KUKA KRL program: EPS_2_251806_MH44A_A_20260213065139.src

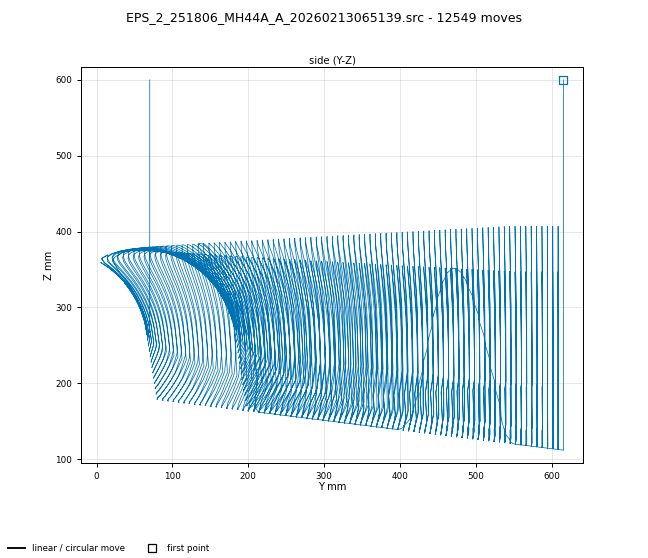
[picture p0: tool path of EPS_2_251806_MH44A_A_20260213065139.src, 12549 of 12551 moves have a stored position in this frame; points joined in program order, loops and branches not executed]
&ACCESS RVP
&REL 4
&COMMENT QRS 19112012
&PARAM EDITMASK = *
DEF PART()
EXT BAS (BAS_COMMAND :IN,REAL :IN )
INT I
BAS (#INITMOV,0 )

;KUKA QRS Post kuka4.cps  Date:22-06-2017 !

File_ID=3029

QRS_PRE_INIT()

;Init var - Until changes are made in qrs_pre_init
Outlet_Square_prg=0
Inlet_1_Square_prg=0
Inlet_2_Square_prg=0
Inlet_3_Square_prg=0
Inlet_4_Square_prg=0
Inlet_5_Square_prg=0

Outlet_1={X 0.000, Y 546.330, Z 306.500, B 0.000, E1 0.000 }
Inlet_1={X 0.000, Y 550.600, Z 246.500, B 0.000, E1 143.000 }
Outlet_1_type=201
Inlet_1_type=201
;QRS#1=Sidecore dimensions
;QRS#2=200-8" PVC SDR 35
;QRS#3=200-8" PVC SDR 35
;QRS#4=
;QRS#5=
;QRS#6=
;QRS#7=
;QRS#8=
;QRS#9=12-08 PSX
;QRS#10=12-08 PSX
;QRS#11=
;QRS#12=
;QRS#13=
;QRS#14=
;QRS#15=
;QRS#16=1220x127x686 2,25'
;QRS#17=EPS Height
;QRS#18=407
;QRS#19=*
;QRS#20= UPDATED VERSION 22-06-2017
;QRS#21=*
Outlet_Square=0100
Inlet_1_Square=0100
Inlet_2_Square=0
Inlet_3_Square=0
Inlet_4_Square=0
Inlet_5_Square=0
Mill_Square=1
Outlet_Square_Prg=204
Inlet_1_Square_prg=204

QRS_INIT()

$ADVANCE=5

; T1
PTP {E1 173.612,E2 173.612}
PTP {X 0,Y 615.492,A -85,B 0,C 180,E1 173.612,E2 173.612,E3 0,E4 0,E5 0,E6 0}
QRS_SPEED_INIT()
LIN {X 0,Y 615.492,Z 600,A -85,B 0,C 180,E1 173.612,E2 173.612,E3 0,E4 0,E5 0,E6 0} C_VEL
LIN {X 0,Y 615.492,Z 121.868,A -85,B 0,C 180,E1 173.612,E2 173.612} C_VEL
LIN {X 0,Y 615.492,Z 113.694,A -85,B 0,C 180,E1 173.612,E2 173.612} C_VEL
LIN {X 0,Y 615.479,Z 111.694,A -85,B 0,C 180,E1 173.426,E2 173.426} C_VEL
LIN {X 0,Y 615.482,Z 111.693,A -85,B 0,C 180,E1 170.801,E2 170.801} C_VEL
LIN {X 0,Y 615.486,Z 111.683,A -85,B 0,C 180,E1 168.139,E2 168.139} C_VEL
LIN {X 0,Y 615.484,Z 111.697,A -85,B 0,C 180,E1 165.451,E2 165.451} C_VEL
LIN {X 0,Y 615.48,Z 111.688,A -85,B 0,C 180,E1 162.729,E2 162.729} C_VEL
LIN {X 0,Y 615.476,Z 111.689,A -85,B 0,C 180,E1 159.967,E2 159.967} C_VEL
LIN {X 0,Y 615.483,Z 111.694,A -85,B 0,C 180,E1 157.155,E2 157.155} C_VEL
LIN {X 0,Y 615.481,Z 111.685,A -85,B 0,C 180,E1 154.284,E2 154.284} C_VEL
LIN {X 0,Y 615.497,Z 111.699,A -85,B 0,C 180,E1 151.547,E2 151.547} C_VEL
LIN {X 0,Y 615.486,Z 111.685,A -85,B 0,C 180,E1 148.914,E2 148.914} C_VEL
LIN {X 0,Y 615.481,Z 111.685,A -85,B 0,C 180,E1 146.466,E2 146.466} C_VEL
LIN {X 0,Y 615.476,Z 111.89,A -85,B 0,C 180,E1 144.275,E2 144.275} C_VEL
LIN {X 0,Y 615.459,Z 125.994,A -85,B 0,C 180,E1 141.721,E2 141.721} C_VEL
LIN {X 0,Y 615.449,Z 136.857,A -85,B 0,C 180,E1 139.801,E2 139.801} C_VEL
LIN {X 0,Y 615.471,Z 242.607,A -85,B 0,C 180,E1 138.549,E2 138.549} C_VEL
LIN {X 0,Y 615.463,Z 255.824,A -85,B 0,C 180,E1 138.261,E2 138.261} C_VEL
LIN {X 0,Y 615.479,Z 268.338,A -85,B 0,C 180,E1 137.853,E2 137.853} C_VEL
LIN {X 0,Y 615.488,Z 280.768,A -85,B 0,C 180,E1 137.3,E2 137.3} C_VEL
LIN {X 0,Y 615.491,Z 291.829,A -85,B 0,C 180,E1 136.662,E2 136.662} C_VEL
LIN {X 0,Y 615.498,Z 303.025,A -85,B 0,C 180,E1 135.852,E2 135.852} C_VEL
LIN {X 0,Y 615.498,Z 311.775,A -85,B 0,C 180,E1 135.067,E2 135.067} C_VEL
LIN {X 0,Y 615.497,Z 320.148,A -85,B 0,C 180,E1 134.148,E2 134.148} C_VEL
LIN {X 0,Y 615.496,Z 328.22,A -85,B 0,C 180,E1 133.048,E2 133.048} C_VEL
LIN {X 0,Y 615.494,Z 333.829,A -85,B 0,C 180,E1 132.081,E2 132.081} C_VEL
LIN {X 0,Y 615.494,Z 338.344,A -85,B 0,C 180,E1 131.095,E2 131.095} C_VEL
LIN {X 0,Y 615.495,Z 341.838,A -85,B 0,C 180,E1 130.09,E2 130.09} C_VEL
LIN {X 0,Y 615.495,Z 344.633,A -85,B 0,C 180,E1 128.903,E2 128.903} C_VEL
LIN {X 0,Y 615.496,Z 345.875,A -85,B 0,C 180,E1 128.013,E2 128.013} C_VEL
LIN {X 0,Y 615.493,Z 346.388,A -85,B 0,C 180,E1 126.937,E2 126.937} C_VEL
LIN {X 0,Y 615.492,Z 345.803,A -85,B 0,C 180,E1 125.834,E2 125.834} C_VEL
LIN {X 0,Y 615.496,Z 344.035,A -85,B 0,C 180,E1 124.702,E2 124.702} C_VEL
LIN {X 0,Y 615.494,Z 340.929,A -85,B 0,C 180,E1 123.535,E2 123.535} C_VEL
LIN {X 0,Y 615.496,Z 336.274,A -85,B 0,C 180,E1 122.332,E2 122.332} C_VEL
LIN {X 0,Y 615.496,Z 331.405,A -85,B 0,C 180,E1 121.385,E2 121.385} C_VEL
LIN {X 0,Y 615.493,Z 324.7,A -85,B 0,C 180,E1 120.349,E2 120.349} C_VEL
LIN {X 0,Y 615.497,Z 317.096,A -85,B 0,C 180,E1 119.406,E2 119.406} C_VEL
LIN {X 0,Y 615.499,Z 307.636,A -85,B 0,C 180,E1 118.452,E2 118.452} C_VEL
LIN {X 0,Y 615.497,Z 297.512,A -85,B 0,C 180,E1 117.637,E2 117.637} C_VEL
LIN {X 0,Y 615.468,Z 286.009,A -85,B 0,C 180,E1 116.893,E2 116.893} C_VEL
LIN {X 0,Y 615.492,Z 274.399,A -85,B 0,C 180,E1 116.307,E2 116.307} C_VEL
LIN {X 0,Y 615.485,Z 262.555,A -85,B 0,C 180,E1 115.852,E2 115.852} C_VEL
LIN {X 0,Y 615.491,Z 249.578,A -85,B 0,C 180,E1 115.497,E2 115.497} C_VEL
LIN {X 0,Y 615.492,Z 236.736,A -85,B 0,C 180,E1 115.28,E2 115.28} C_VEL
LIN {X 0,Y 615.464,Z 136.666,A -85,B 0,C 180,E1 114.105,E2 114.105} C_VEL
LIN {X 0,Y 615.49,Z 121.785,A -85,B 0,C 180,E1 111.432,E2 111.432} C_VEL
LIN {X 0,Y 615.49,Z 111.686,A -85,B 0,C 180,E1 109.598,E2 109.598} C_VEL
LIN {X 0,Y 615.468,Z 111.687,A -85,B 0,C 180,E1 107.271,E2 107.271} C_VEL
LIN {X 0,Y 615.474,Z 111.697,A -85,B 0,C 180,E1 104.549,E2 104.549} C_VEL
LIN {X 0,Y 615.488,Z 111.688,A -85,B 0,C 180,E1 101.861,E2 101.861} C_VEL
LIN {X 0,Y 615.459,Z 111.69,A -85,B 0,C 180,E1 99.199,E2 99.199} C_VEL
LIN {X 0,Y 615.492,Z 111.699,A -85,B 0,C 180,E1 96.557,E2 96.557} C_VEL
LIN {X 0,Y 615.487,Z 111.686,A -85,B 0,C 180,E1 93.928,E2 93.928} C_VEL
LIN {X 0,Y 615.459,Z 111.691,A -85,B 0,C 180,E1 91.309,E2 91.309} C_VEL
LIN {X 0,Y 615.492,Z 111.702,A -85,B 0,C 180,E1 88.691,E2 88.691} C_VEL
LIN {X 0,Y 615.486,Z 111.685,A -85,B 0,C 180,E1 86.071,E2 86.071} C_VEL
LIN {X 0,Y 615.461,Z 111.692,A -85,B 0,C 180,E1 83.443,E2 83.443} C_VEL
LIN {X 0,Y 615.492,Z 111.699,A -85,B 0,C 180,E1 80.801,E2 80.801} C_VEL
LIN {X 0,Y 615.483,Z 111.685,A -85,B 0,C 180,E1 78.139,E2 78.139} C_VEL
LIN {X 0,Y 615.466,Z 111.694,A -85,B 0,C 180,E1 75.451,E2 75.451} C_VEL
LIN {X 0,Y 615.489,Z 111.691,A -85,B 0,C 180,E1 72.73,E2 72.73} C_VEL
LIN {X 0,Y 615.465,Z 111.688,A -85,B 0,C 180,E1 69.967,E2 69.967} C_VEL
LIN {X 0,Y 615.467,Z 111.694,A -85,B 0,C 180,E1 67.659,E2 67.659} C_VEL
LIN {X 0,Y 615.488,Z 111.693,A -85,B 0,C 180,E1 65.008,E2 65.008} C_VEL
LIN {X 0,Y 615.465,Z 111.689,A -85,B 0,C 180,E1 62.084,E2 62.084} C_VEL
LIN {X 0,Y 615.468,Z 111.694,A -85,B 0,C 180,E1 59.839,E2 59.839} C_VEL
LIN {X 0,Y 615.488,Z 111.7,A -85,B 0,C 180,E1 57.543,E2 57.543} C_VEL
LIN {X 0,Y 615.488,Z 111.692,A -85,B 0,C 180,E1 55.185,E2 55.185} C_VEL
LIN {X 0,Y 615.491,Z 111.683,A -85,B 0,C 180,E1 52.758,E2 52.758} C_VEL
LIN {X 0,Y 615.475,Z 111.697,A -85,B 0,C 180,E1 49.912,E2 49.912} C_VEL
LIN {X 0,Y 615.488,Z 111.684,A -85,B 0,C 180,E1 46.952,E2 46.952} C_VEL
LIN {X 0,Y 615.469,Z 111.695,A -85,B 0,C 180,E1 44.151,E2 44.151} C_VEL
LIN {X 0,Y 615.486,Z 111.691,A -85,B 0,C 180,E1 41.474,E2 41.474} C_VEL
LIN {X 0,Y 615.48,Z 111.684,A -85,B 0,C 180,E1 38.905,E2 38.905} C_VEL
LIN {X 0,Y 615.47,Z 111.693,A -85,B 0,C 180,E1 36.426,E2 36.426} C_VEL
LIN {X 0,Y 615.486,Z 111.688,A -85,B 0,C 180,E1 33.534,E2 33.534} C_VEL
LIN {X 0,Y 615.472,Z 111.687,A -85,B 0,C 180,E1 30.92,E2 30.92} C_VEL
LIN {X 0,Y 615.479,Z 111.696,A -85,B 0,C 180,E1 28.449,E2 28.449} C_VEL
LIN {X 0,Y 615.488,Z 111.685,A -85,B 0,C 180,E1 25.57,E2 25.57} C_VEL
LIN {X 0,Y 615.47,Z 111.691,A -85,B 0,C 180,E1 22.845,E2 22.845} C_VEL
LIN {X 0,Y 615.485,Z 111.697,A -85,B 0,C 180,E1 20.557,E2 20.557} C_VEL
LIN {X 0,Y 615.484,Z 111.689,A -85,B 0,C 180,E1 17.957,E2 17.957} C_VEL
LIN {X 0,Y 615.473,Z 111.688,A -85,B 0,C 180,E1 15.226,E2 15.226} C_VEL
LIN {X 0,Y 615.49,Z 111.7,A -85,B 0,C 180,E1 12.53,E2 12.53} C_VEL
LIN {X 0,Y 615.494,Z 111.682,A -85,B 0,C 180,E1 9.862,E2 9.862} C_VEL
LIN {X 0,Y 615.472,Z 111.691,A -85,B 0,C 180,E1 7.216,E2 7.216} C_VEL
LIN {X 0,Y 615.488,Z 111.696,A -85,B 0,C 180,E1 4.584,E2 4.584} C_VEL
LIN {X 0,Y 615.5,Z 111.68,A -85,B 0,C 180,E1 1.963,E2 1.963} C_VEL
LIN {X 0,Y 615.474,Z 111.692,A -85,B 0,C 180,E1 -0.654,E2 -0.654} C_VEL
LIN {X 0,Y 615.485,Z 111.695,A -85,B 0,C 180,E1 -3.273,E2 -3.273} C_VEL
LIN {X 0,Y 615.497,Z 111.681,A -85,B 0,C 180,E1 -5.899,E2 -5.899} C_VEL
LIN {X 0,Y 615.474,Z 111.694,A -85,B 0,C 180,E1 -8.537,E2 -8.537} C_VEL
LIN {X 0,Y 615.482,Z 111.692,A -85,B 0,C 180,E1 -11.193,E2 -11.193} C_VEL
LIN {X 0,Y 615.482,Z 111.685,A -85,B 0,C 180,E1 -13.932,E2 -13.932} C_VEL
LIN {X 0,Y 615.491,Z 111.698,A -85,B 0,C 180,E1 -16.587,E2 -16.587} C_VEL
LIN {X 0,Y 615.485,Z 111.685,A -85,B 0,C 180,E1 -19.338,E2 -19.338} C_VEL
LIN {X 0,Y 615.477,Z 111.692,A -85,B 0,C 180,E1 -22.137,E2 -22.137} C_VEL
LIN {X 0,Y 615.479,Z 111.689,A -85,B 0,C 180,E1 -24.992,E2 -24.992} C_VEL
LIN {X 0,Y 615.484,Z 111.685,A -85,B 0,C 180,E1 -27.178,E2 -27.178} C_VEL
LIN {X 0,Y 615.477,Z 111.689,A -85,B 0,C 180,E1 -29.794,E2 -29.794} C_VEL
LIN {X 0,Y 615.485,Z 111.698,A -85,B 0,C 180,E1 -32.458,E2 -32.458} C_VEL
LIN {X 0,Y 615.479,Z 111.688,A -85,B 0,C 180,E1 -34.816,E2 -34.816} C_VEL
LIN {X 0,Y 615.492,Z 111.682,A -85,B 0,C 180,E1 -37.242,E2 -37.242} C_VEL
LIN {X 0,Y 615.496,Z 111.701,A -85,B 0,C 180,E1 -40.09,E2 -40.09} C_VEL
LIN {X 0,Y 615.488,Z 111.683,A -85,B 0,C 180,E1 -43.048,E2 -43.048} C_VEL
LIN {X 0,Y 615.488,Z 111.701,A -85,B 0,C 180,E1 -46.003,E2 -46.003} C_VEL
LIN {X 0,Y 615.487,Z 111.683,A -85,B 0,C 180,E1 -48.906,E2 -48.906} C_VEL
LIN {X 0,Y 615.49,Z 111.698,A -85,B 0,C 180,E1 -51.932,E2 -51.932} C_VEL
LIN {X 0,Y 615.474,Z 111.689,A -85,B 0,C 180,E1 -54.383,E2 -54.383} C_VEL
LIN {X 0,Y 615.487,Z 111.683,A -85,B 0,C 180,E1 -56.764,E2 -56.764} C_VEL
LIN {X 0,Y 615.481,Z 111.688,A -85,B 0,C 180,E1 -59.08,E2 -59.08} C_VEL
LIN {X 0,Y 615.498,Z 111.7,A -85,B 0,C 180,E1 -61.548,E2 -61.548} C_VEL
LIN {X 0,Y 615.485,Z 111.683,A -85,B 0,C 180,E1 -64.432,E2 -64.432} C_VEL
LIN {X 0,Y 615.488,Z 111.874,A -85,B 0,C 180,E1 -66.711,E2 -66.711} C_VEL
LIN {X 0,Y 615.45,Z 133.105,A -85,B 0,C 180,E1 -69.453,E2 -69.453} C_VEL
LIN {X 0,Y 615.494,Z 154.836,A -85,B 0,C 180,E1 -72.215,E2 -72.215} C_VEL
LIN {X 0,Y 615.485,Z 176.625,A -85,B 0,C 180,E1 -74.943,E2 -74.943} C_VEL
LIN {X 0,Y 615.449,Z 194.136,A -85,B 0,C 180,E1 -77.113,E2 -77.113} C_VEL
LIN {X 0,Y 615.488,Z 302.833,A -85,B 0,C 180,E1 -78.411,E2 -78.411} C_VEL
LIN {X 0,Y 615.477,Z 315.347,A -85,B 0,C 180,E1 -78.682,E2 -78.682} C_VEL
LIN {X 0,Y 615.488,Z 328.618,A -85,B 0,C 180,E1 -79.113,E2 -79.113} C_VEL
LIN {X 0,Y 615.477,Z 340.479,A -85,B 0,C 180,E1 -79.639,E2 -79.639} C_VEL
LIN {X 0,Y 615.494,Z 351.994,A -85,B 0,C 180,E1 -80.304,E2 -80.304} C_VEL
LIN {X 0,Y 615.499,Z 362.341,A -85,B 0,C 180,E1 -81.05,E2 -81.05} C_VEL
LIN {X 0,Y 615.497,Z 370.812,A -85,B 0,C 180,E1 -81.794,E2 -81.794} C_VEL
LIN {X 0,Y 615.498,Z 378.606,A -85,B 0,C 180,E1 -82.62,E2 -82.62} C_VEL
LIN {X 0,Y 615.496,Z 386.203,A -85,B 0,C 180,E1 -83.608,E2 -83.608} C_VEL
LIN {X 0,Y 615.498,Z 393.205,A -85,B 0,C 180,E1 -84.759,E2 -84.759} C_VEL
LIN {X 0,Y 615.494,Z 397.851,A -85,B 0,C 180,E1 -85.744,E2 -85.744} C_VEL
LIN {X 0,Y 615.494,Z 401.399,A -85,B 0,C 180,E1 -86.727,E2 -86.727} C_VEL
LIN {X 0,Y 615.497,Z 403.233,A -85,B 0,C 180,E1 -87.382,E2 -87.382} C_VEL
LIN {X 0,Y 615.5,Z 404.607,A -85,B 0,C 180,E1 -88.037,E2 -88.037} C_VEL
LIN {X 0,Y 615.496,Z 406.173,A -85,B 0,C 180,E1 -89.346,E2 -89.346} C_VEL
LIN {X 0,Y 615.494,Z 406.389,A -85,B 0,C 180,E1 -90,E2 -90} C_VEL
LIN {X 0,Y 615.495,Z 405.58,A -85,B 0,C 180,E1 -91.309,E2 -91.309} C_VEL
LIN {X 0,Y 615.5,Z 404.607,A -85,B 0,C 180,E1 -91.963,E2 -91.963} C_VEL
LIN {X 0,Y 615.497,Z 403.233,A -85,B 0,C 180,E1 -92.618,E2 -92.618} C_VEL
LIN {X 0,Y 615.496,Z 400.35,A -85,B 0,C 180,E1 -93.601,E2 -93.601} C_VEL
LIN {X 0,Y 615.498,Z 396.442,A -85,B 0,C 180,E1 -94.584,E2 -94.584} C_VEL
LIN {X 0,Y 615.499,Z 391.405,A -85,B 0,C 180,E1 -95.57,E2 -95.57} C_VEL
LIN {X 0,Y 615.497,Z 384.87,A -85,B 0,C 180,E1 -96.583,E2 -96.583} C_VEL
LIN {X 0,Y 615.497,Z 377.134,A -85,B 0,C 180,E1 -97.545,E2 -97.545} C_VEL
LIN {X 0,Y 615.498,Z 369.046,A -85,B 0,C 180,E1 -98.371,E2 -98.371} C_VEL
LIN {X 0,Y 615.499,Z 359.169,A -85,B 0,C 180,E1 -99.199,E2 -99.199} C_VEL
LIN {X 0,Y 615.488,Z 347.983,A -85,B 0,C 180,E1 -99.945,E2 -99.945} C_VEL
LIN {X 0,Y 615.482,Z 337.025,A -85,B 0,C 180,E1 -100.527,E2 -100.527} C_VEL
LIN {X 0,Y 615.48,Z 324.492,A -85,B 0,C 180,E1 -101.04,E2 -101.04} C_VEL
LIN {X 0,Y 615.479,Z 312.071,A -85,B 0,C 180,E1 -101.402,E2 -101.402} C_VEL
LIN {X 0,Y 615.493,Z 298.472,A -85,B 0,C 180,E1 -101.652,E2 -101.652} C_VEL
LIN {X 0,Y 615.449,Z 194.137,A -85,B 0,C 180,E1 -102.887,E2 -102.887} C_VEL
LIN {X 0,Y 615.493,Z 171.176,A -85,B 0,C 180,E1 -105.735,E2 -105.735} C_VEL
LIN {X 0,Y 615.469,Z 149.687,A -85,B 0,C 180,E1 -108.436,E2 -108.436} C_VEL
LIN {X 0,Y 615.496,Z 127.568,A -85,B 0,C 180,E1 -111.256,E2 -111.256} C_VEL
LIN {X 0,Y 615.49,Z 111.683,A -85,B 0,C 180,E1 -113.333,E2 -113.333} C_VEL
LIN {X 0,Y 615.48,Z 111.685,A -85,B 0,C 180,E1 -115.716,E2 -115.716} C_VEL
LIN {X 0,Y 615.497,Z 111.701,A -85,B 0,C 180,E1 -118.451,E2 -118.451} C_VEL
LIN {X 0,Y 615.486,Z 111.685,A -85,B 0,C 180,E1 -121.085,E2 -121.085} C_VEL
LIN {X 0,Y 615.48,Z 111.685,A -85,B 0,C 180,E1 -123.533,E2 -123.533} C_VEL
LIN {X 0,Y 615.489,Z 111.697,A -85,B 0,C 180,E1 -126.424,E2 -126.424} C_VEL
LIN {X 0,Y 615.495,Z 111.681,A -85,B 0,C 180,E1 -129.063,E2 -129.063} C_VEL
LIN {X 0,Y 615.495,Z 111.699,A -85,B 0,C 180,E1 -132.081,E2 -132.081} C_VEL
LIN {X 0,Y 615.494,Z 111.681,A -85,B 0,C 180,E1 -135.068,E2 -135.068} C_VEL
LIN {X 0,Y 615.489,Z 111.699,A -85,B 0,C 180,E1 -137.919,E2 -137.919} C_VEL
LIN {X 0,Y 615.494,Z 111.681,A -85,B 0,C 180,E1 -140.937,E2 -140.937} C_VEL
LIN {X 0,Y 615.479,Z 111.694,A -85,B 0,C 180,E1 -143.574,E2 -143.574} C_VEL
LIN {X 0,Y 615.484,Z 111.686,A -85,B 0,C 180,E1 -146.466,E2 -146.466} C_VEL
LIN {X 0,Y 615.476,Z 111.687,A -85,B 0,C 180,E1 -149.079,E2 -149.079} C_VEL
LIN {X 0,Y 615.488,Z 111.697,A -85,B 0,C 180,E1 -151.549,E2 -151.549} C_VEL
LIN {X 0,Y 615.486,Z 111.684,A -85,B 0,C 180,E1 -154.431,E2 -154.431} C_VEL
LIN {X 0,Y 615.474,Z 111.693,A -85,B 0,C 180,E1 -157.155,E2 -157.155} C_VEL
LIN {X 0,Y 615.492,Z 111.699,A -85,B 0,C 180,E1 -159.441,E2 -159.441} C_VEL
LIN {X 0,Y 615.479,Z 111.688,A -85,B 0,C 180,E1 -162.043,E2 -162.043} C_VEL
LIN {X 0,Y 615.476,Z 111.688,A -85,B 0,C 180,E1 -164.774,E2 -164.774} C_VEL
LIN {X 0,Y 615.491,Z 111.697,A -85,B 0,C 180,E1 -167.47,E2 -167.47} C_VEL
LIN {X 0,Y 615.494,Z 111.682,A -85,B 0,C 180,E1 -170.138,E2 -170.138} C_VEL
LIN {X 0,Y 615.476,Z 111.692,A -85,B 0,C 180,E1 -172.784,E2 -172.784} C_VEL
LIN {X 0,Y 615.485,Z 111.695,A -85,B 0,C 180,E1 -175.415,E2 -175.415} C_VEL
LIN {X 0,Y 615.5,Z 111.68,A -85,B 0,C 180,E1 -178.037,E2 -178.037} C_VEL
LIN {X 0,Y 615.475,Z 111.693,A -85,B 0,C 180,E1 -180.654,E2 -180.654} C_VEL
LIN {X 0,Y 615.483,Z 111.694,A -85,B 0,C 180,E1 -183.273,E2 -183.273} C_VEL
LIN {X 0,Y 615.497,Z 111.68,A -85,B 0,C 180,E1 -185.898,E2 -185.898} C_VEL
LIN {X 0,Y 615.479,Z 111.694,A -85,B 0,C 180,E1 -186.574,E2 -186.574} C_VEL
LIN {X 0,Y 614.805,Z 111.843,A -85,B 0,C 180,E1 -187.12,E2 -187.12} C_VEL
LIN {X 0,Y 611.97,Z 112.249,A -85,B 0,C 180,E1 -188.006,E2 -188.006} C_VEL
LIN {X 0,Y 609.579,Z 112.562,A -85,B 0,C 180,E1 -188.719,E2 -188.719} C_VEL
LIN {X 0,Y 608.547,Z 112.68,A -85,B 0,C 180,E1 -189.269,E2 -189.269} C_VEL
LIN {X 0,Y 608.459,Z 112.688,A -85,B 0,C 180,E1 -189.455,E2 -189.455} C_VEL
LIN {X 0,Y 608.46,Z 112.687,A -85,B 0,C 180,E1 -192,E2 -192} C_VEL
LIN {X 0,Y 608.472,Z 112.696,A -85,B 0,C 180,E1 -194.72,E2 -194.72} C_VEL
LIN {X 0,Y 608.446,Z 112.689,A -85,B 0,C 180,E1 -197.477,E2 -197.477} C_VEL
LIN {X 0,Y 608.458,Z 112.692,A -85,B 0,C 180,E1 -200.274,E2 -200.274} C_VEL
LIN {X 0,Y 608.456,Z 112.697,A -85,B 0,C 180,E1 -202.476,E2 -202.476} C_VEL
LIN {X 0,Y 608.449,Z 112.688,A -85,B 0,C 180,E1 -205.301,E2 -205.301} C_VEL
LIN {X 0,Y 608.444,Z 112.689,A -85,B 0,C 180,E1 -207.518,E2 -207.518} C_VEL
LIN {X 0,Y 608.459,Z 112.691,A -85,B 0,C 180,E1 -209.971,E2 -209.971} C_VEL
LIN {X 0,Y 608.464,Z 112.693,A -85,B 0,C 180,E1 -212.523,E2 -212.523} C_VEL
LIN {X 0,Y 608.436,Z 112.69,A -85,B 0,C 180,E1 -215.278,E2 -215.278} C_VEL
LIN {X 0,Y 608.469,Z 112.882,A -85,B 0,C 180,E1 -215.682,E2 -215.682} C_VEL
LIN {X 0,Y 608.454,Z 126.888,A -85,B 0,C 180,E1 -218.239,E2 -218.239} C_VEL
LIN {X 0,Y 608.41,Z 136.835,A -85,B 0,C 180,E1 -220.036,E2 -220.036} C_VEL
LIN {X 0,Y 608.566,Z 209.469,A -85,B 0,C 180,E1 -220.911,E2 -220.911} C_VEL
LIN {X 0,Y 608.527,Z 243.725,A -85,B 0,C 180,E1 -221.336,E2 -221.336} C_VEL
LIN {X 0,Y 608.498,Z 257.197,A -85,B 0,C 180,E1 -221.643,E2 -221.643} C_VEL
LIN {X 0,Y 608.518,Z 269.405,A -85,B 0,C 180,E1 -222.056,E2 -222.056} C_VEL
LIN {X 0,Y 608.498,Z 281.583,A -85,B 0,C 180,E1 -222.615,E2 -222.615} C_VEL
LIN {X 0,Y 608.481,Z 293.329,A -85,B 0,C 180,E1 -223.31,E2 -223.31} C_VEL
LIN {X 0,Y 608.471,Z 303.556,A -85,B 0,C 180,E1 -224.067,E2 -224.067} C_VEL
LIN {X 0,Y 608.459,Z 313.651,A -85,B 0,C 180,E1 -225,E2 -225} C_VEL
LIN {X 0,Y 608.465,Z 321.857,A -85,B 0,C 180,E1 -225.933,E2 -225.933} C_VEL
LIN {X 0,Y 608.448,Z 328.564,A -85,B 0,C 180,E1 -226.868,E2 -226.868} C_VEL
LIN {X 0,Y 608.429,Z 334.691,A -85,B 0,C 180,E1 -227.936,E2 -227.936} C_VEL
LIN {X 0,Y 608.431,Z 338.725,A -85,B 0,C 180,E1 -228.822,E2 -228.822} C_VEL
LIN {X 0,Y 608.435,Z 343.094,A -85,B 0,C 180,E1 -230.128,E2 -230.128} C_VEL
LIN {X 0,Y 608.415,Z 345.781,A -85,B 0,C 180,E1 -231.408,E2 -231.408} C_VEL
LIN {X 0,Y 608.428,Z 346.691,A -85,B 0,C 180,E1 -232.251,E2 -232.251} C_VEL
LIN {X 0,Y 608.429,Z 346.997,A -85,B 0,C 180,E1 -233.084,E2 -233.084} C_VEL
LIN {X 0,Y 608.42,Z 346.607,A -85,B 0,C 180,E1 -233.958,E2 -233.958} C_VEL
LIN {X 0,Y 608.423,Z 345.089,A -85,B 0,C 180,E1 -235.098,E2 -235.098} C_VEL
LIN {X 0,Y 608.435,Z 342.045,A -85,B 0,C 180,E1 -236.328,E2 -236.328} C_VEL
LIN {X 0,Y 608.428,Z 337.808,A -85,B 0,C 180,E1 -237.482,E2 -237.482} C_VEL
LIN {X 0,Y 608.453,Z 331.568,A -85,B 0,C 180,E1 -238.731,E2 -238.731} C_VEL
LIN {X 0,Y 608.444,Z 324.761,A -85,B 0,C 180,E1 -239.774,E2 -239.774} C_VEL
LIN {X 0,Y 608.451,Z 316.481,A -85,B 0,C 180,E1 -240.79,E2 -240.79} C_VEL
LIN {X 0,Y 608.467,Z 306.918,A -85,B 0,C 180,E1 -241.734,E2 -241.734} C_VEL
LIN {X 0,Y 608.479,Z 296.237,A -85,B 0,C 180,E1 -242.58,E2 -242.58} C_VEL
LIN {X 0,Y 608.464,Z 286.143,A -85,B 0,C 180,E1 -243.227,E2 -243.227} C_VEL
LIN {X 0,Y 608.509,Z 274.25,A -85,B 0,C 180,E1 -243.829,E2 -243.829} C_VEL
LIN {X 0,Y 608.524,Z 261.875,A -85,B 0,C 180,E1 -244.303,E2 -244.303} C_VEL
LIN {X 0,Y 608.549,Z 249.13,A -85,B 0,C 180,E1 -244.649,E2 -244.649} C_VEL
LIN {X 0,Y 608.55,Z 236.184,A -85,B 0,C 180,E1 -244.864,E2 -244.864} C_VEL
LIN {X 0,Y 608.43,Z 136.897,A -85,B 0,C 180,E1 -246.042,E2 -246.042} C_VEL
LIN {X 0,Y 608.485,Z 122.406,A -85,B 0,C 180,E1 -248.665,E2 -248.665} C_VEL
LIN {X 0,Y 608.472,Z 112.687,A -85,B 0,C 180,E1 -250.474,E2 -250.474} C_VEL
LIN {X 0,Y 608.469,Z 112.691,A -85,B 0,C 180,E1 -253.471,E2 -253.471} C_VEL
LIN {X 0,Y 608.476,Z 112.69,A -85,B 0,C 180,E1 -255.98,E2 -255.98} C_VEL
LIN {X 0,Y 608.432,Z 112.69,A -85,B 0,C 180,E1 -258.676,E2 -258.676} C_VEL
LIN {X 0,Y 608.45,Z 112.695,A -85,B 0,C 180,E1 -261.364,E2 -261.364} C_VEL
LIN {X 0,Y 608.494,Z 112.685,A -85,B 0,C 180,E1 -264.033,E2 -264.033} C_VEL
LIN {X 0,Y 608.454,Z 112.688,A -85,B 0,C 180,E1 -266.689,E2 -266.689} C_VEL
LIN {X 0,Y 608.481,Z 112.694,A -85,B 0,C 180,E1 -269.338,E2 -269.338} C_VEL
LIN {X 0,Y 608.469,Z 112.687,A -85,B 0,C 180,E1 -271.986,E2 -271.986} C_VEL
LIN {X 0,Y 608.432,Z 112.692,A -85,B 0,C 180,E1 -274.638,E2 -274.638} C_VEL
LIN {X 0,Y 608.432,Z 112.692,A -85,B 0,C 180,E1 -276.633,E2 -276.633} C_VEL
LIN {X 0,Y 608.475,Z 112.692,A -85,B 0,C 180,E1 -279.306,E2 -279.306} C_VEL
LIN {X 0,Y 608.455,Z 112.687,A -85,B 0,C 180,E1 -282,E2 -282} C_VEL
LIN {X 0,Y 608.464,Z 112.692,A -85,B 0,C 180,E1 -284.721,E2 -284.721} C_VEL
LIN {X 0,Y 608.45,Z 112.69,A -85,B 0,C 180,E1 -287.477,E2 -287.477} C_VEL
LIN {X 0,Y 608.448,Z 112.69,A -85,B 0,C 180,E1 -290.275,E2 -290.275} C_VEL
LIN {X 0,Y 608.459,Z 112.692,A -85,B 0,C 180,E1 -292.476,E2 -292.476} C_VEL
LIN {X 0,Y 608.451,Z 112.69,A -85,B 0,C 180,E1 -295.301,E2 -295.301} C_VEL
LIN {X 0,Y 608.443,Z 112.689,A -85,B 0,C 180,E1 -297.518,E2 -297.518} C_VEL
LIN {X 0,Y 608.451,Z 112.689,A -85,B 0,C 180,E1 -299.969,E2 -299.969} C_VEL
LIN {X 0,Y 608.462,Z 112.697,A -85,B 0,C 180,E1 -302.523,E2 -302.523} C_VEL
LIN {X 0,Y 608.435,Z 112.69,A -85,B 0,C 180,E1 -305.278,E2 -305.278} C_VEL
LIN {X 0,Y 608.461,Z 112.688,A -85,B 0,C 180,E1 -307.747,E2 -307.747} C_VEL
LIN {X 0,Y 608.447,Z 112.699,A -85,B 0,C 180,E1 -310.329,E2 -310.329} C_VEL
LIN {X 0,Y 608.456,Z 112.688,A -85,B 0,C 180,E1 -312.959,E2 -312.959} C_VEL
LIN {X 0,Y 608.443,Z 112.692,A -85,B 0,C 180,E1 -315.737,E2 -315.737} C_VEL
LIN {X 0,Y 608.459,Z 112.693,A -85,B 0,C 180,E1 -317.939,E2 -317.939} C_VEL
LIN {X 0,Y 608.479,Z 112.686,A -85,B 0,C 180,E1 -320.701,E2 -320.701} C_VEL
LIN {X 0,Y 608.45,Z 112.688,A -85,B 0,C 180,E1 -323.085,E2 -323.085} C_VEL
LIN {X 0,Y 608.461,Z 112.69,A -85,B 0,C 180,E1 -325.53,E2 -325.53} C_VEL
LIN {X 0,Y 608.462,Z 112.697,A -85,B 0,C 180,E1 -327.905,E2 -327.905} C_VEL
LIN {X 0,Y 608.469,Z 112.69,A -85,B 0,C 180,E1 -330.221,E2 -330.221} C_VEL
LIN {X 0,Y 608.472,Z 112.685,A -85,B 0,C 180,E1 -332.793,E2 -332.793} C_VEL
LIN {X 0,Y 608.449,Z 112.694,A -85,B 0,C 180,E1 -335.429,E2 -335.429} C_VEL
LIN {X 0,Y 608.472,Z 112.686,A -85,B 0,C 180,E1 -338.309,E2 -338.309} C_VEL
LIN {X 0,Y 608.469,Z 112.691,A -85,B 0,C 180,E1 -341.284,E2 -341.284} C_VEL
LIN {X 0,Y 608.461,Z 112.69,A -85,B 0,C 180,E1 -343.906,E2 -343.906} C_VEL
LIN {X 0,Y 608.454,Z 112.688,A -85,B 0,C 180,E1 -346.643,E2 -346.643} C_VEL
LIN {X 0,Y 608.463,Z 112.697,A -85,B 0,C 180,E1 -349.35,E2 -349.35} C_VEL
LIN {X 0,Y 608.479,Z 112.685,A -85,B 0,C 180,E1 -352.033,E2 -352.033} C_VEL
LIN {X 0,Y 608.454,Z 112.69,A -85,B 0,C 180,E1 -354.698,E2 -354.698} C_VEL
LIN {X 0,Y 608.473,Z 112.692,A -85,B 0,C 180,E1 -357.352,E2 -357.352} C_VEL
LIN {X 0,Y 608.477,Z 112.685,A -85,B 0,C 180,E1 -360,E2 -360} C_VEL
LIN {X 0,Y 608.467,Z 112.69,A -85,B 0,C 180,E1 -362.648,E2 -362.648} C_VEL
LIN {X 0,Y 608.464,Z 112.691,A -85,B 0,C 180,E1 -365.302,E2 -365.302} C_VEL
LIN {X 0,Y 608.476,Z 112.685,A -85,B 0,C 180,E1 -367.967,E2 -367.967} C_VEL
LIN {X 0,Y 608.461,Z 112.694,A -85,B 0,C 180,E1 -370.65,E2 -370.65} C_VEL
LIN {X 0,Y 608.46,Z 112.688,A -85,B 0,C 180,E1 -373.357,E2 -373.357} C_VEL
LIN {X 0,Y 608.457,Z 112.689,A -85,B 0,C 180,E1 -376.094,E2 -376.094} C_VEL
LIN {X 0,Y 608.457,Z 112.693,A -85,B 0,C 180,E1 -378.87,E2 -378.87} C_VEL
LIN {X 0,Y 608.469,Z 112.686,A -85,B 0,C 180,E1 -381.692,E2 -381.692} C_VEL
LIN {X 0,Y 608.45,Z 112.697,A -85,B 0,C 180,E1 -384.571,E2 -384.571} C_VEL
LIN {X 0,Y 608.477,Z 112.685,A -85,B 0,C 180,E1 -387.208,E2 -387.208} C_VEL
LIN {X 0,Y 608.462,Z 112.691,A -85,B 0,C 180,E1 -389.971,E2 -389.971} C_VEL
LIN {X 0,Y 608.458,Z 112.689,A -85,B 0,C 180,E1 -392.88,E2 -392.88} C_VEL
LIN {X 0,Y 608.436,Z 112.69,A -85,B 0,C 180,E1 -395.278,E2 -395.278} C_VEL
LIN {X 0,Y 608.473,Z 112.689,A -85,B 0,C 180,E1 -397.746,E2 -397.746} C_VEL
LIN {X 0,Y 608.453,Z 112.694,A -85,B 0,C 180,E1 -400.329,E2 -400.329} C_VEL
LIN {X 0,Y 608.454,Z 112.687,A -85,B 0,C 180,E1 -402.96,E2 -402.96} C_VEL
LIN {X 0,Y 608.461,Z 112.693,A -85,B 0,C 180,E1 -405.736,E2 -405.736} C_VEL
LIN {X 0,Y 608.458,Z 112.687,A -85,B 0,C 180,E1 -408.659,E2 -408.659} C_VEL
LIN {X 0,Y 608.47,Z 112.689,A -85,B 0,C 180,E1 -411.412,E2 -411.412} C_VEL
LIN {X 0,Y 608.446,Z 112.695,A -85,B 0,C 180,E1 -413.955,E2 -413.955} C_VEL
LIN {X 0,Y 608.448,Z 112.69,A -85,B 0,C 180,E1 -416.329,E2 -416.329} C_VEL
LIN {X 0,Y 608.448,Z 112.688,A -85,B 0,C 180,E1 -418.733,E2 -418.733} C_VEL
LIN {X 0,Y 608.478,Z 112.692,A -85,B 0,C 180,E1 -421.38,E2 -421.38} C_VEL
LIN {X 0,Y 608.468,Z 112.686,A -85,B 0,C 180,E1 -424.28,E2 -424.28} C_VEL
LIN {X 0,Y 608.467,Z 112.727,A -85,B 0,C 180,E1 -426.539,E2 -426.539} C_VEL
LIN {X 0,Y 608.595,Z 127.568,A -85,B 0,C 180,E1 -428.491,E2 -428.491} C_VEL
LIN {X 0,Y 608.498,Z 149.174,A -85,B 0,C 180,E1 -431.277,E2 -431.277} C_VEL
LIN {X 0,Y 608.495,Z 168.579,A -85,B 0,C 180,E1 -433.744,E2 -433.744} C_VEL
LIN {X 0,Y 608.479,Z 190.346,A -85,B 0,C 180,E1 -436.474,E2 -436.474} C_VEL
LIN {X 0,Y 608.446,Z 194.355,A -85,B 0,C 180,E1 -436.972,E2 -436.972} C_VEL
LIN {X 0,Y 608.546,Z 302.949,A -85,B 0,C 180,E1 -438.277,E2 -438.277} C_VEL
LIN {X 0,Y 608.512,Z 316.218,A -85,B 0,C 180,E1 -438.572,E2 -438.572} C_VEL
LIN {X 0,Y 608.514,Z 328.629,A -85,B 0,C 180,E1 -438.982,E2 -438.982} C_VEL
LIN {X 0,Y 608.499,Z 340.635,A -85,B 0,C 180,E1 -439.519,E2 -439.519} C_VEL
LIN {X 0,Y 608.484,Z 352.198,A -85,B 0,C 180,E1 -440.191,E2 -440.191} C_VEL
LIN {X 0,Y 608.485,Z 362.594,A -85,B 0,C 180,E1 -440.946,E2 -440.946} C_VEL
LIN {X 0,Y 608.475,Z 371.112,A -85,B 0,C 180,E1 -441.699,E2 -441.699} C_VEL
LIN {X 0,Y 608.471,Z 378.96,A -85,B 0,C 180,E1 -442.534,E2 -442.534} C_VEL
LIN {X 0,Y 608.461,Z 386.287,A -85,B 0,C 180,E1 -443.485,E2 -443.485} C_VEL
LIN {X 0,Y 608.451,Z 391.866,A -85,B 0,C 180,E1 -444.366,E2 -444.366} C_VEL
LIN {X 0,Y 608.432,Z 396.95,A -85,B 0,C 180,E1 -445.362,E2 -445.362} C_VEL
LIN {X 0,Y 608.449,Z 400.896,A -85,B 0,C 180,E1 -446.358,E2 -446.358} C_VEL
LIN {X 0,Y 608.425,Z 403.809,A -85,B 0,C 180,E1 -447.352,E2 -447.352} C_VEL
LIN {X 0,Y 608.445,Z 405.201,A -85,B 0,C 180,E1 -448.014,E2 -448.014} C_VEL
LIN {X 0,Y 608.438,Z 406.783,A -85,B 0,C 180,E1 -449.338,E2 -449.338} C_VEL
LIN {X 0,Y 608.434,Z 407,A -85,B 0,C 180,E1 -450,E2 -450} C_VEL
LIN {X 0,Y 608.448,Z 406.184,A -85,B 0,C 180,E1 -451.324,E2 -451.324} C_VEL
LIN {X 0,Y 608.445,Z 405.201,A -85,B 0,C 180,E1 -451.986,E2 -451.986} C_VEL
LIN {X 0,Y 608.425,Z 403.809,A -85,B 0,C 180,E1 -452.648,E2 -452.648} C_VEL
LIN {X 0,Y 608.449,Z 400.896,A -85,B 0,C 180,E1 -453.642,E2 -453.642} C_VEL
LIN {X 0,Y 608.432,Z 396.95,A -85,B 0,C 180,E1 -454.638,E2 -454.638} C_VEL
LIN {X 0,Y 608.438,Z 390.877,A -85,B 0,C 180,E1 -455.801,E2 -455.801} C_VEL
LIN {X 0,Y 608.462,Z 384.236,A -85,B 0,C 180,E1 -456.799,E2 -456.799} C_VEL
LIN {X 0,Y 608.456,Z 375.99,A -85,B 0,C 180,E1 -457.8,E2 -457.8} C_VEL
LIN {X 0,Y 608.472,Z 367.537,A -85,B 0,C 180,E1 -458.636,E2 -458.636} C_VEL
LIN {X 0,Y 608.479,Z 357.092,A -85,B 0,C 180,E1 -459.473,E2 -459.473} C_VEL
LIN {X 0,Y 608.489,Z 346.758,A -85,B 0,C 180,E1 -460.145,E2 -460.145} C_VEL
LIN {X 0,Y 608.519,Z 335.268,A -85,B 0,C 180,E1 -460.74,E2 -460.74} C_VEL
LIN {X 0,Y 608.528,Z 322.893,A -85,B 0,C 180,E1 -461.225,E2 -461.225} C_VEL
LIN {X 0,Y 608.544,Z 309.443,A -85,B 0,C 180,E1 -461.597,E2 -461.597} C_VEL
LIN {X 0,Y 608.552,Z 297.092,A -85,B 0,C 180,E1 -461.808,E2 -461.808} C_VEL
LIN {X 0,Y 608.434,Z 194.27,A -85,B 0,C 180,E1 -463.038,E2 -463.038} C_VEL
LIN {X 0,Y 608.523,Z 171.24,A -85,B 0,C 180,E1 -465.92,E2 -465.92} C_VEL
LIN {X 0,Y 608.53,Z 150.97,A -85,B 0,C 180,E1 -468.492,E2 -468.492} C_VEL
LIN {X 0,Y 608.571,Z 130.298,A -85,B 0,C 180,E1 -471.154,E2 -471.154} C_VEL
LIN {X 0,Y 608.52,Z 112.898,A -85,B 0,C 180,E1 -473.436,E2 -473.436} C_VEL
LIN {X 0,Y 608.459,Z 112.69,A -85,B 0,C 180,E1 -473.845,E2 -473.845} C_VEL
LIN {X 0,Y 608.443,Z 112.692,A -85,B 0,C 180,E1 -476.035,E2 -476.035} C_VEL
LIN {X 0,Y 608.477,Z 112.692,A -85,B 0,C 180,E1 -478.62,E2 -478.62} C_VEL
LIN {X 0,Y 608.446,Z 112.688,A -85,B 0,C 180,E1 -481.317,E2 -481.317} C_VEL
LIN {X 0,Y 608.473,Z 112.687,A -85,B 0,C 180,E1 -483.735,E2 -483.735} C_VEL
LIN {X 0,Y 608.446,Z 112.696,A -85,B 0,C 180,E1 -486.092,E2 -486.092} C_VEL
LIN {X 0,Y 608.47,Z 112.69,A -85,B 0,C 180,E1 -488.588,E2 -488.588} C_VEL
LIN {X 0,Y 608.457,Z 112.687,A -85,B 0,C 180,E1 -491.341,E2 -491.341} C_VEL
LIN {X 0,Y 608.464,Z 112.694,A -85,B 0,C 180,E1 -494.264,E2 -494.264} C_VEL
LIN {X 0,Y 608.453,Z 112.687,A -85,B 0,C 180,E1 -497.04,E2 -497.04} C_VEL
LIN {X 0,Y 608.452,Z 112.693,A -85,B 0,C 180,E1 -499.696,E2 -499.696} C_VEL
LIN {X 0,Y 608.471,Z 112.69,A -85,B 0,C 180,E1 -502.254,E2 -502.254} C_VEL
LIN {X 0,Y 608.442,Z 112.689,A -85,B 0,C 180,E1 -505.095,E2 -505.095} C_VEL
LIN {X 0,Y 608.467,Z 112.694,A -85,B 0,C 180,E1 -507.905,E2 -507.905} C_VEL
LIN {X 0,Y 608.466,Z 112.689,A -85,B 0,C 180,E1 -510.22,E2 -510.22} C_VEL
LIN {X 0,Y 608.475,Z 112.685,A -85,B 0,C 180,E1 -512.793,E2 -512.793} C_VEL
LIN {X 0,Y 608.452,Z 112.695,A -85,B 0,C 180,E1 -515.429,E2 -515.429} C_VEL
LIN {X 0,Y 608.471,Z 112.686,A -85,B 0,C 180,E1 -518.308,E2 -518.308} C_VEL
LIN {X 0,Y 608.473,Z 112.692,A -85,B 0,C 180,E1 -521.282,E2 -521.282} C_VEL
LIN {X 0,Y 608.46,Z 112.689,A -85,B 0,C 180,E1 -523.906,E2 -523.906} C_VEL
LIN {X 0,Y 608.455,Z 112.688,A -85,B 0,C 180,E1 -526.643,E2 -526.643} C_VEL
LIN {X 0,Y 608.464,Z 112.696,A -85,B 0,C 180,E1 -529.35,E2 -529.35} C_VEL
LIN {X 0,Y 608.478,Z 112.685,A -85,B 0,C 180,E1 -532.033,E2 -532.033} C_VEL
LIN {X 0,Y 608.457,Z 112.69,A -85,B 0,C 180,E1 -534.698,E2 -534.698} C_VEL
LIN {X 0,Y 608.475,Z 112.691,A -85,B 0,C 180,E1 -537.352,E2 -537.352} C_VEL
LIN {X 0,Y 608.477,Z 112.684,A -85,B 0,C 180,E1 -540,E2 -540} C_VEL
LIN {X 0,Y 608.469,Z 112.69,A -85,B 0,C 180,E1 -542.648,E2 -542.648} C_VEL
LIN {X 0,Y 608.463,Z 112.691,A -85,B 0,C 180,E1 -545.302,E2 -545.302} C_VEL
LIN {X 0,Y 608.476,Z 112.685,A -85,B 0,C 180,E1 -547.967,E2 -547.967} C_VEL
LIN {X 0,Y 608.459,Z 112.688,A -85,B 0,C 180,E1 -549.455,E2 -549.455} C_VEL
LIN {X 0,Y 607.783,Z 112.773,A -85,B 0,C 180,E1 -550.007,E2 -550.007} C_VEL
LIN {X 0,Y 604.929,Z 113.135,A -85,B 0,C 180,E1 -550.904,E2 -550.904} C_VEL
LIN {X 0,Y 602.524,Z 113.43,A -85,B 0,C 180,E1 -551.626,E2 -551.626} C_VEL
LIN {X 0,Y 601.491,Z 113.557,A -85,B 0,C 180,E1 -552.182,E2 -552.182} C_VEL
LIN {X 0,Y 601.407,Z 113.568,A -85,B 0,C 180,E1 -552.371,E2 -552.371} C_VEL
LIN {X 0,Y 601.426,Z 113.57,A -85,B 0,C 180,E1 -554.897,E2 -554.897} C_VEL
LIN {X 0,Y 601.431,Z 113.567,A -85,B 0,C 180,E1 -556.986,E2 -556.986} C_VEL
LIN {X 0,Y 601.402,Z 113.566,A -85,B 0,C 180,E1 -559.809,E2 -559.809} C_VEL
LIN {X 0,Y 601.413,Z 113.575,A -85,B 0,C 180,E1 -562.606,E2 -562.606} C_VEL
LIN {X 0,Y 601.4,Z 113.571,A -85,B 0,C 180,E1 -564.879,E2 -564.879} C_VEL
LIN {X 0,Y 601.419,Z 113.566,A -85,B 0,C 180,E1 -567.867,E2 -567.867} C_VEL
LIN {X 0,Y 601.425,Z 113.57,A -85,B 0,C 180,E1 -570.164,E2 -570.164} C_VEL
LIN {X 0,Y 601.424,Z 113.567,A -85,B 0,C 180,E1 -572.716,E2 -572.716} C_VEL
LIN {X 0,Y 601.434,Z 113.673,A -85,B 0,C 180,E1 -575.62,E2 -575.62} C_VEL
LIN {X 0,Y 601.415,Z 126.853,A -85,B 0,C 180,E1 -578.055,E2 -578.055} C_VEL
LIN {X 0,Y 601.371,Z 136.851,A -85,B 0,C 180,E1 -579.884,E2 -579.884} C_VEL
LIN {X 0,Y 601.643,Z 143.323,A -85,B 0,C 180,E1 -579.976,E2 -579.976} C_VEL
LIN {X 0,Y 601.591,Z 243.395,A -85,B 0,C 180,E1 -581.193,E2 -581.193} C_VEL
LIN {X 0,Y 601.563,Z 256.881,A -85,B 0,C 180,E1 -581.501,E2 -581.501} C_VEL
LIN {X 0,Y 601.533,Z 269.327,A -85,B 0,C 180,E1 -581.924,E2 -581.924} C_VEL
LIN {X 0,Y 601.495,Z 280.541,A -85,B 0,C 180,E1 -582.436,E2 -582.436} C_VEL
LIN {X 0,Y 601.468,Z 292.224,A -85,B 0,C 180,E1 -583.122,E2 -583.122} C_VEL
LIN {X 0,Y 601.458,Z 303.182,A -85,B 0,C 180,E1 -583.931,E2 -583.931} C_VEL
LIN {X 0,Y 601.408,Z 312.206,A -85,B 0,C 180,E1 -584.754,E2 -584.754} C_VEL
LIN {X 0,Y 601.39,Z 320.768,A -85,B 0,C 180,E1 -585.713,E2 -585.713} C_VEL
LIN {X 0,Y 601.376,Z 327.644,A -85,B 0,C 180,E1 -586.656,E2 -586.656} C_VEL
LIN {X 0,Y 601.37,Z 334.433,A -85,B 0,C 180,E1 -587.823,E2 -587.823} C_VEL
LIN {X 0,Y 601.333,Z 338.707,A -85,B 0,C 180,E1 -588.767,E2 -588.767} C_VEL
LIN {X 0,Y 601.343,Z 342.846,A -85,B 0,C 180,E1 -590,E2 -590} C_VEL
LIN {X 0,Y 601.314,Z 344.894,A -85,B 0,C 180,E1 -590.866,E2 -590.866} C_VEL
LIN {X 0,Y 601.329,Z 346.208,A -85,B 0,C 180,E1 -591.726,E2 -591.726} C_VEL
LIN {X 0,Y 601.331,Z 346.91,A -85,B 0,C 180,E1 -592.631,E2 -592.631} C_VEL
LIN {X 0,Y 601.313,Z 346.759,A -85,B 0,C 180,E1 -593.751,E2 -593.751} C_VEL
LIN {X 0,Y 601.335,Z 345.187,A -85,B 0,C 180,E1 -595.063,E2 -595.063} C_VEL
LIN {X 0,Y 601.327,Z 342.875,A -85,B 0,C 180,E1 -596.079,E2 -596.079} C_VEL
LIN {X 0,Y 601.334,Z 338.81,A -85,B 0,C 180,E1 -597.297,E2 -597.297} C_VEL
LIN {X 0,Y 601.355,Z 334.416,A -85,B 0,C 180,E1 -598.271,E2 -598.271} C_VEL
LIN {X 0,Y 601.383,Z 328.847,A -85,B 0,C 180,E1 -599.251,E2 -599.251} C_VEL
LIN {X 0,Y 601.381,Z 322.028,A -85,B 0,C 180,E1 -600.22,E2 -600.22} C_VEL
LIN {X 0,Y 601.396,Z 313.339,A -85,B 0,C 180,E1 -601.218,E2 -601.218} C_VEL
LIN {X 0,Y 601.448,Z 303.49,A -85,B 0,C 180,E1 -602.134,E2 -602.134} C_VEL
LIN {X 0,Y 601.469,Z 293.395,A -85,B 0,C 180,E1 -602.89,E2 -602.89} C_VEL
LIN {X 0,Y 601.491,Z 282.524,A -85,B 0,C 180,E1 -603.547,E2 -603.547} C_VEL
LIN {X 0,Y 601.527,Z 270.689,A -85,B 0,C 180,E1 -604.11,E2 -604.11} C_VEL
LIN {X 0,Y 601.59,Z 258.162,A -85,B 0,C 180,E1 -604.552,E2 -604.552} C_VEL
LIN {X 0,Y 601.615,Z 245.689,A -85,B 0,C 180,E1 -604.854,E2 -604.854} C_VEL
LIN {X 0,Y 601.62,Z 227.279,A -85,B 0,C 180,E1 -605.108,E2 -605.108} C_VEL
LIN {X 0,Y 601.508,Z 137.822,A -85,B 0,C 180,E1 -606.183,E2 -606.183} C_VEL
LIN {X 0,Y 601.423,Z 136.742,A -85,B 0,C 180,E1 -606.225,E2 -606.225} C_VEL
LIN {X 0,Y 601.421,Z 120.505,A -85,B 0,C 180,E1 -609.204,E2 -609.204} C_VEL
LIN {X 0,Y 601.457,Z 113.562,A -85,B 0,C 180,E1 -610.504,E2 -610.504} C_VEL
LIN {X 0,Y 601.438,Z 113.572,A -85,B 0,C 180,E1 -613.713,E2 -613.713} C_VEL
LIN {X 0,Y 601.407,Z 113.566,A -85,B 0,C 180,E1 -616.484,E2 -616.484} C_VEL
LIN {X 0,Y 601.409,Z 113.569,A -85,B 0,C 180,E1 -619.224,E2 -619.224} C_VEL
LIN {X 0,Y 601.441,Z 113.565,A -85,B 0,C 180,E1 -621.939,E2 -621.939} C_VEL
LIN {X 0,Y 601.412,Z 113.565,A -85,B 0,C 180,E1 -624.636,E2 -624.636} C_VEL
LIN {X 0,Y 601.445,Z 113.569,A -85,B 0,C 180,E1 -627.321,E2 -627.321} C_VEL
LIN {X 0,Y 601.446,Z 113.562,A -85,B 0,C 180,E1 -630,E2 -630} C_VEL
LIN {X 0,Y 601.423,Z 113.565,A -85,B 0,C 180,E1 -632.679,E2 -632.679} C_VEL
LIN {X 0,Y 601.437,Z 113.569,A -85,B 0,C 180,E1 -635.364,E2 -635.364} C_VEL
LIN {X 0,Y 601.436,Z 113.562,A -85,B 0,C 180,E1 -638.061,E2 -638.061} C_VEL
LIN {X 0,Y 601.42,Z 113.573,A -85,B 0,C 180,E1 -641.01,E2 -641.01} C_VEL
LIN {X 0,Y 601.415,Z 113.567,A -85,B 0,C 180,E1 -643.516,E2 -643.516} C_VEL
LIN {X 0,Y 601.426,Z 113.564,A -85,B 0,C 180,E1 -646.287,E2 -646.287} C_VEL
LIN {X 0,Y 601.416,Z 113.57,A -85,B 0,C 180,E1 -649.099,E2 -649.099} C_VEL
LIN {X 0,Y 601.409,Z 113.569,A -85,B 0,C 180,E1 -651.239,E2 -651.239} C_VEL
LIN {X 0,Y 601.44,Z 113.563,A -85,B 0,C 180,E1 -654.141,E2 -654.141} C_VEL
LIN {X 0,Y 601.452,Z 113.563,A -85,B 0,C 180,E1 -657.111,E2 -657.111} C_VEL
LIN {X 0,Y 601.413,Z 113.565,A -85,B 0,C 180,E1 -659.393,E2 -659.393} C_VEL
LIN {X 0,Y 601.403,Z 113.566,A -85,B 0,C 180,E1 -661.727,E2 -661.727} C_VEL
LIN {X 0,Y 601.418,Z 113.568,A -85,B 0,C 180,E1 -664.119,E2 -664.119} C_VEL
LIN {X 0,Y 601.436,Z 113.562,A -85,B 0,C 180,E1 -667.382,E2 -667.382} C_VEL
LIN {X 0,Y 601.4,Z 113.571,A -85,B 0,C 180,E1 -669.996,E2 -669.996} C_VEL
LIN {X 0,Y 601.415,Z 113.568,A -85,B 0,C 180,E1 -672.67,E2 -672.67} C_VEL
LIN {X 0,Y 601.425,Z 113.564,A -85,B 0,C 180,E1 -675.482,E2 -675.482} C_VEL
LIN {X 0,Y 601.423,Z 113.569,A -85,B 0,C 180,E1 -678.407,E2 -678.407} C_VEL
LIN {X 0,Y 601.437,Z 113.562,A -85,B 0,C 180,E1 -680.876,E2 -680.876} C_VEL
LIN {X 0,Y 601.405,Z 113.571,A -85,B 0,C 180,E1 -683.739,E2 -683.739} C_VEL
LIN {X 0,Y 601.426,Z 113.563,A -85,B 0,C 180,E1 -686.687,E2 -686.687} C_VEL
LIN {X 0,Y 601.42,Z 113.564,A -85,B 0,C 180,E1 -689.058,E2 -689.058} C_VEL
LIN {X 0,Y 601.423,Z 113.567,A -85,B 0,C 180,E1 -691.373,E2 -691.373} C_VEL
LIN {X 0,Y 601.398,Z 113.575,A -85,B 0,C 180,E1 -693.636,E2 -693.636} C_VEL
LIN {X 0,Y 601.458,Z 113.567,A -85,B 0,C 180,E1 -695.86,E2 -695.86} C_VEL
LIN {X 0,Y 601.406,Z 113.565,A -85,B 0,C 180,E1 -698.761,E2 -698.761} C_VEL
LIN {X 0,Y 601.419,Z 113.574,A -85,B 0,C 180,E1 -701.608,E2 -701.608} C_VEL
LIN {X 0,Y 601.408,Z 113.565,A -85,B 0,C 180,E1 -704.409,E2 -704.409} C_VEL
LIN {X 0,Y 601.418,Z 113.57,A -85,B 0,C 180,E1 -707.172,E2 -707.172} C_VEL
LIN {X 0,Y 601.438,Z 113.563,A -85,B 0,C 180,E1 -709.905,E2 -709.905} C_VEL
LIN {X 0,Y 601.435,Z 113.563,A -85,B 0,C 180,E1 -712.615,E2 -712.615} C_VEL
LIN {X 0,Y 601.423,Z 113.572,A -85,B 0,C 180,E1 -715.308,E2 -715.308} C_VEL
LIN {X 0,Y 601.438,Z 113.562,A -85,B 0,C 180,E1 -717.991,E2 -717.991} C_VEL
LIN {X 0,Y 601.442,Z 113.565,A -85,B 0,C 180,E1 -720.67,E2 -720.67} C_VEL
LIN {X 0,Y 601.43,Z 113.567,A -85,B 0,C 180,E1 -723.35,E2 -723.35} C_VEL
LIN {X 0,Y 601.438,Z 113.561,A -85,B 0,C 180,E1 -726.037,E2 -726.037} C_VEL
LIN {X 0,Y 601.409,Z 113.573,A -85,B 0,C 180,E1 -728.738,E2 -728.738} C_VEL
LIN {X 0,Y 601.433,Z 113.563,A -85,B 0,C 180,E1 -731.458,E2 -731.458} C_VEL
LIN {X 0,Y 601.418,Z 113.566,A -85,B 0,C 180,E1 -734.206,E2 -734.206} C_VEL
LIN {X 0,Y 601.431,Z 113.567,A -85,B 0,C 180,E1 -736.986,E2 -736.986} C_VEL
LIN {X 0,Y 601.403,Z 113.566,A -85,B 0,C 180,E1 -739.81,E2 -739.81} C_VEL
LIN {X 0,Y 601.414,Z 113.574,A -85,B 0,C 180,E1 -742.606,E2 -742.606} C_VEL
LIN {X 0,Y 601.4,Z 113.57,A -85,B 0,C 180,E1 -744.879,E2 -744.879} C_VEL
LIN {X 0,Y 601.413,Z 113.564,A -85,B 0,C 180,E1 -747.363,E2 -747.363} C_VEL
LIN {X 0,Y 601.427,Z 113.57,A -85,B 0,C 180,E1 -750.164,E2 -750.164} C_VEL
LIN {X 0,Y 601.422,Z 113.567,A -85,B 0,C 180,E1 -752.716,E2 -752.716} C_VEL
LIN {X 0,Y 601.392,Z 113.567,A -85,B 0,C 180,E1 -755.112,E2 -755.112} C_VEL
LIN {X 0,Y 601.437,Z 113.562,A -85,B 0,C 180,E1 -757.419,E2 -757.419} C_VEL
LIN {X 0,Y 601.411,Z 113.573,A -85,B 0,C 180,E1 -759.995,E2 -759.995} C_VEL
LIN {X 0,Y 601.411,Z 113.566,A -85,B 0,C 180,E1 -762.671,E2 -762.671} C_VEL
LIN {X 0,Y 601.427,Z 113.566,A -85,B 0,C 180,E1 -765.482,E2 -765.482} C_VEL
LIN {X 0,Y 601.424,Z 113.566,A -85,B 0,C 180,E1 -768.407,E2 -768.407} C_VEL
LIN {X 0,Y 601.437,Z 113.561,A -85,B 0,C 180,E1 -770.876,E2 -770.876} C_VEL
LIN {X 0,Y 601.403,Z 113.57,A -85,B 0,C 180,E1 -773.417,E2 -773.417} C_VEL
LIN {X 0,Y 601.433,Z 113.566,A -85,B 0,C 180,E1 -776.065,E2 -776.065} C_VEL
LIN {X 0,Y 601.421,Z 113.564,A -85,B 0,C 180,E1 -778.546,E2 -778.546} C_VEL
LIN {X 0,Y 601.437,Z 113.569,A -85,B 0,C 180,E1 -781.374,E2 -781.374} C_VEL
LIN {X 0,Y 601.402,Z 113.575,A -85,B 0,C 180,E1 -783.636,E2 -783.636} C_VEL
LIN {X 0,Y 601.428,Z 113.58,A -85,B 0,C 180,E1 -786.362,E2 -786.362} C_VEL
LIN {X 0,Y 601.75,Z 116.65,A -85,B 0,C 180,E1 -786.786,E2 -786.786} C_VEL
LIN {X 0,Y 601.612,Z 138.486,A -85,B 0,C 180,E1 -789.663,E2 -789.663} C_VEL
LIN {X 0,Y 601.549,Z 160.322,A -85,B 0,C 180,E1 -792.492,E2 -792.492} C_VEL
LIN {X 0,Y 601.46,Z 180.793,A -85,B 0,C 180,E1 -795.104,E2 -795.104} C_VEL
LIN {X 0,Y 601.42,Z 194.355,A -85,B 0,C 180,E1 -796.818,E2 -796.818} C_VEL
LIN {X 0,Y 601.63,Z 207.668,A -85,B 0,C 180,E1 -796.983,E2 -796.983} C_VEL
LIN {X 0,Y 601.613,Z 302.949,A -85,B 0,C 180,E1 -798.14,E2 -798.14} C_VEL
LIN {X 0,Y 601.56,Z 316.219,A -85,B 0,C 180,E1 -798.438,E2 -798.438} C_VEL
LIN {X 0,Y 601.546,Z 327.904,A -85,B 0,C 180,E1 -798.825,E2 -798.825} C_VEL
LIN {X 0,Y 601.522,Z 340.634,A -85,B 0,C 180,E1 -799.396,E2 -799.396} C_VEL
LIN {X 0,Y 601.483,Z 352.2,A -85,B 0,C 180,E1 -800.076,E2 -800.076} C_VEL
LIN {X 0,Y 601.444,Z 362.596,A -85,B 0,C 180,E1 -800.839,E2 -800.839} C_VEL
LIN {X 0,Y 601.429,Z 371.112,A -85,B 0,C 180,E1 -801.601,E2 -801.601} C_VEL
LIN {X 0,Y 601.418,Z 378.961,A -85,B 0,C 180,E1 -802.446,E2 -802.446} C_VEL
LIN {X 0,Y 601.37,Z 386.225,A -85,B 0,C 180,E1 -803.398,E2 -803.398} C_VEL
LIN {X 0,Y 601.372,Z 391.866,A -85,B 0,C 180,E1 -804.299,E2 -804.299} C_VEL
LIN {X 0,Y 601.336,Z 396.95,A -85,B 0,C 180,E1 -805.307,E2 -805.307} C_VEL
LIN {X 0,Y 601.368,Z 400.896,A -85,B 0,C 180,E1 -806.315,E2 -806.315} C_VEL
LIN {X 0,Y 601.325,Z 403.809,A -85,B 0,C 180,E1 -807.32,E2 -807.32} C_VEL
LIN {X 0,Y 601.343,Z 405.202,A -85,B 0,C 180,E1 -807.991,E2 -807.991} C_VEL
LIN {X 0,Y 601.339,Z 406.784,A -85,B 0,C 180,E1 -809.33,E2 -809.33} C_VEL
LIN {X 0,Y 601.335,Z 407,A -85,B 0,C 180,E1 -810,E2 -810} C_VEL
LIN {X 0,Y 601.347,Z 406.184,A -85,B 0,C 180,E1 -811.339,E2 -811.339} C_VEL
LIN {X 0,Y 601.343,Z 405.202,A -85,B 0,C 180,E1 -812.009,E2 -812.009} C_VEL
LIN {X 0,Y 601.325,Z 403.81,A -85,B 0,C 180,E1 -812.68,E2 -812.68} C_VEL
LIN {X 0,Y 601.368,Z 400.896,A -85,B 0,C 180,E1 -813.685,E2 -813.685} C_VEL
LIN {X 0,Y 601.336,Z 396.95,A -85,B 0,C 180,E1 -814.693,E2 -814.693} C_VEL
LIN {X 0,Y 601.373,Z 390.878,A -85,B 0,C 180,E1 -815.869,E2 -815.869} C_VEL
LIN {X 0,Y 601.382,Z 384.236,A -85,B 0,C 180,E1 -816.88,E2 -816.88} C_VEL
LIN {X 0,Y 601.4,Z 375.99,A -85,B 0,C 180,E1 -817.892,E2 -817.892} C_VEL
LIN {X 0,Y 601.436,Z 367.538,A -85,B 0,C 180,E1 -818.738,E2 -818.738} C_VEL
LIN {X 0,Y 601.449,Z 357.094,A -85,B 0,C 180,E1 -819.585,E2 -819.585} C_VEL
LIN {X 0,Y 601.467,Z 346.76,A -85,B 0,C 180,E1 -820.264,E2 -820.264} C_VEL
LIN {X 0,Y 601.538,Z 334.599,A -85,B 0,C 180,E1 -820.896,E2 -820.896} C_VEL
LIN {X 0,Y 601.555,Z 322.22,A -85,B 0,C 180,E1 -821.379,E2 -821.379} C_VEL
LIN {X 0,Y 601.583,Z 309.442,A -85,B 0,C 180,E1 -821.733,E2 -821.733} C_VEL
LIN {X 0,Y 601.623,Z 297.092,A -85,B 0,C 180,E1 -821.946,E2 -821.946} C_VEL
LIN {X 0,Y 601.531,Z 195.152,A -85,B 0,C 180,E1 -823.169,E2 -823.169} C_VEL
LIN {X 0,Y 601.426,Z 194.27,A -85,B 0,C 180,E1 -823.193,E2 -823.193} C_VEL
LIN {X 0,Y 601.512,Z 171.24,A -85,B 0,C 180,E1 -826.11,E2 -826.11} C_VEL
LIN {X 0,Y 601.575,Z 151.699,A -85,B 0,C 180,E1 -828.619,E2 -828.619} C_VEL
LIN {X 0,Y 601.667,Z 130.298,A -85,B 0,C 180,E1 -831.409,E2 -831.409} C_VEL
LIN {X 0,Y 601.749,Z 115.286,A -85,B 0,C 180,E1 -833.397,E2 -833.397} C_VEL
LIN {X 0,Y 601.421,Z 113.568,A -85,B 0,C 180,E1 -833.661,E2 -833.661} C_VEL
LIN {X 0,Y 601.402,Z 113.575,A -85,B 0,C 180,E1 -836.364,E2 -836.364} C_VEL
LIN {X 0,Y 601.441,Z 113.566,A -85,B 0,C 180,E1 -838.789,E2 -838.789} C_VEL
LIN {X 0,Y 601.421,Z 113.564,A -85,B 0,C 180,E1 -841.454,E2 -841.454} C_VEL
LIN {X 0,Y 601.428,Z 113.57,A -85,B 0,C 180,E1 -844.118,E2 -844.118} C_VEL
LIN {X 0,Y 601.438,Z 113.562,A -85,B 0,C 180,E1 -847.382,E2 -847.382} C_VEL
LIN {X 0,Y 601.411,Z 113.572,A -85,B 0,C 180,E1 -849.995,E2 -849.995} C_VEL
LIN {X 0,Y 601.412,Z 113.567,A -85,B 0,C 180,E1 -852.67,E2 -852.67} C_VEL
LIN {X 0,Y 601.426,Z 113.565,A -85,B 0,C 180,E1 -855.482,E2 -855.482} C_VEL
LIN {X 0,Y 601.424,Z 113.567,A -85,B 0,C 180,E1 -858.406,E2 -858.406} C_VEL
LIN {X 0,Y 601.437,Z 113.561,A -85,B 0,C 180,E1 -860.875,E2 -860.875} C_VEL
LIN {X 0,Y 601.401,Z 113.569,A -85,B 0,C 180,E1 -863.417,E2 -863.417} C_VEL
LIN {X 0,Y 601.431,Z 113.568,A -85,B 0,C 180,E1 -866.064,E2 -866.064} C_VEL
LIN {X 0,Y 601.429,Z 113.563,A -85,B 0,C 180,E1 -868.543,E2 -868.543} C_VEL
LIN {X 0,Y 601.429,Z 113.567,A -85,B 0,C 180,E1 -871.373,E2 -871.373} C_VEL
LIN {X 0,Y 601.402,Z 113.576,A -85,B 0,C 180,E1 -873.636,E2 -873.636} C_VEL
LIN {X 0,Y 601.456,Z 113.565,A -85,B 0,C 180,E1 -875.859,E2 -875.859} C_VEL
LIN {X 0,Y 601.408,Z 113.566,A -85,B 0,C 180,E1 -878.761,E2 -878.761} C_VEL
LIN {X 0,Y 601.421,Z 113.572,A -85,B 0,C 180,E1 -881.608,E2 -881.608} C_VEL
LIN {X 0,Y 601.409,Z 113.565,A -85,B 0,C 180,E1 -884.408,E2 -884.408} C_VEL
LIN {X 0,Y 601.419,Z 113.571,A -85,B 0,C 180,E1 -887.172,E2 -887.172} C_VEL
LIN {X 0,Y 601.438,Z 113.563,A -85,B 0,C 180,E1 -889.905,E2 -889.905} C_VEL
LIN {X 0,Y 601.436,Z 113.563,A -85,B 0,C 180,E1 -892.615,E2 -892.615} C_VEL
LIN {X 0,Y 601.42,Z 113.571,A -85,B 0,C 180,E1 -895.308,E2 -895.308} C_VEL
LIN {X 0,Y 601.438,Z 113.562,A -85,B 0,C 180,E1 -897.991,E2 -897.991} C_VEL
LIN {X 0,Y 601.442,Z 113.565,A -85,B 0,C 180,E1 -900.669,E2 -900.669} C_VEL
LIN {X 0,Y 601.428,Z 113.567,A -85,B 0,C 180,E1 -903.349,E2 -903.349} C_VEL
LIN {X 0,Y 601.438,Z 113.561,A -85,B 0,C 180,E1 -906.037,E2 -906.037} C_VEL
LIN {X 0,Y 601.411,Z 113.573,A -85,B 0,C 180,E1 -908.738,E2 -908.738} C_VEL
LIN {X 0,Y 601.432,Z 113.563,A -85,B 0,C 180,E1 -911.458,E2 -911.458} C_VEL
LIN {X 0,Y 601.407,Z 113.568,A -85,B 0,C 180,E1 -912.371,E2 -912.371} C_VEL
LIN {X 0,Y 600.741,Z 113.658,A -85,B 0,C 180,E1 -912.93,E2 -912.93} C_VEL
LIN {X 0,Y 597.891,Z 114.013,A -85,B 0,C 180,E1 -913.838,E2 -913.838} C_VEL
LIN {X 0,Y 595.481,Z 114.311,A -85,B 0,C 180,E1 -914.568,E2 -914.568} C_VEL
LIN {X 0,Y 594.444,Z 114.437,A -85,B 0,C 180,E1 -915.132,E2 -915.132} C_VEL
LIN {X 0,Y 594.358,Z 114.445,A -85,B 0,C 180,E1 -915.323,E2 -915.323} C_VEL
LIN {X 0,Y 594.387,Z 114.442,A -85,B 0,C 180,E1 -917.193,E2 -917.193} C_VEL
LIN {X 0,Y 594.373,Z 114.444,A -85,B 0,C 180,E1 -920.054,E2 -920.054} C_VEL
LIN {X 0,Y 594.361,Z 114.447,A -85,B 0,C 180,E1 -922.967,E2 -922.967} C_VEL
LIN {X 0,Y 594.374,Z 114.443,A -85,B 0,C 180,E1 -925.193,E2 -925.193} C_VEL
LIN {X 0,Y 594.383,Z 114.441,A -85,B 0,C 180,E1 -927.527,E2 -927.527} C_VEL
LIN {X 0,Y 594.384,Z 114.45,A -85,B 0,C 180,E1 -930.328,E2 -930.328} C_VEL
LIN {X 0,Y 594.378,Z 114.443,A -85,B 0,C 180,E1 -932.95,E2 -932.95} C_VEL
LIN {X 0,Y 594.397,Z 114.496,A -85,B 0,C 180,E1 -935.562,E2 -935.562} C_VEL
LIN {X 0,Y 594.396,Z 127.206,A -85,B 0,C 180,E1 -937.94,E2 -937.94} C_VEL
LIN {X 0,Y 594.345,Z 136.803,A -85,B 0,C 180,E1 -939.717,E2 -939.717} C_VEL
LIN {X 0,Y 594.722,Z 141.55,A -85,B 0,C 180,E1 -939.8,E2 -939.8} C_VEL
LIN {X 0,Y 594.647,Z 242.907,A -85,B 0,C 180,E1 -941.043,E2 -941.043} C_VEL
LIN {X 0,Y 594.625,Z 255.991,A -85,B 0,C 180,E1 -941.339,E2 -941.339} C_VEL
LIN {X 0,Y 594.573,Z 268.151,A -85,B 0,C 180,E1 -941.747,E2 -941.747} C_VEL
LIN {X 0,Y 594.518,Z 280.204,A -85,B 0,C 180,E1 -942.292,E2 -942.292} C_VEL
LIN {X 0,Y 594.48,Z 291.89,A -85,B 0,C 180,E1 -942.982,E2 -942.982} C_VEL
LIN {X 0,Y 594.42,Z 302.047,A -85,B 0,C 180,E1 -943.73,E2 -943.73} C_VEL
LIN {X 0,Y 594.384,Z 310.885,A -85,B 0,C 180,E1 -944.524,E2 -944.524} C_VEL
LIN {X 0,Y 594.331,Z 319.584,A -85,B 0,C 180,E1 -945.477,E2 -945.477} C_VEL
LIN {X 0,Y 594.303,Z 326.668,A -85,B 0,C 180,E1 -946.432,E2 -946.432} C_VEL
LIN {X 0,Y 594.289,Z 333.689,A -85,B 0,C 180,E1 -947.618,E2 -947.618} C_VEL
LIN {X 0,Y 594.244,Z 337.906,A -85,B 0,C 180,E1 -948.525,E2 -948.525} C_VEL
LIN {X 0,Y 594.25,Z 341.236,A -85,B 0,C 180,E1 -949.424,E2 -949.424} C_VEL
LIN {X 0,Y 594.225,Z 343.745,A -85,B 0,C 180,E1 -950.308,E2 -950.308} C_VEL
LIN {X 0,Y 594.207,Z 345.698,A -85,B 0,C 180,E1 -951.317,E2 -951.317} C_VEL
LIN {X 0,Y 594.226,Z 346.815,A -85,B 0,C 180,E1 -952.412,E2 -952.412} C_VEL
LIN {X 0,Y 594.23,Z 346.767,A -85,B 0,C 180,E1 -953.747,E2 -953.747} C_VEL
LIN {X 0,Y 594.222,Z 345.825,A -85,B 0,C 180,E1 -954.694,E2 -954.694} C_VEL
LIN {X 0,Y 594.247,Z 343.488,A -85,B 0,C 180,E1 -955.88,E2 -955.88} C_VEL
LIN {X 0,Y 594.254,Z 339.703,A -85,B 0,C 180,E1 -957.107,E2 -957.107} C_VEL
LIN {X 0,Y 594.273,Z 335.35,A -85,B 0,C 180,E1 -958.137,E2 -958.137} C_VEL
LIN {X 0,Y 594.305,Z 329.364,A -85,B 0,C 180,E1 -959.239,E2 -959.239} C_VEL
LIN {X 0,Y 594.305,Z 322.691,A -85,B 0,C 180,E1 -960.22,E2 -960.22} C_VEL
LIN {X 0,Y 594.347,Z 314.276,A -85,B 0,C 180,E1 -961.217,E2 -961.217} C_VEL
LIN {X 0,Y 594.404,Z 304.507,A -85,B 0,C 180,E1 -962.155,E2 -962.155} C_VEL
LIN {X 0,Y 594.46,Z 294.62,A -85,B 0,C 180,E1 -962.925,E2 -962.925} C_VEL
LIN {X 0,Y 594.498,Z 282.63,A -85,B 0,C 180,E1 -963.666,E2 -963.666} C_VEL
LIN {X 0,Y 594.547,Z 270.444,A -85,B 0,C 180,E1 -964.252,E2 -964.252} C_VEL
LIN {X 0,Y 594.608,Z 257.759,A -85,B 0,C 180,E1 -964.701,E2 -964.701} C_VEL
LIN {X 0,Y 594.671,Z 244.969,A -85,B 0,C 180,E1 -965.008,E2 -965.008} C_VEL
LIN {X 0,Y 594.668,Z 221.418,A -85,B 0,C 180,E1 -965.322,E2 -965.322} C_VEL
LIN {X 0,Y 594.613,Z 138.561,A -85,B 0,C 180,E1 -966.329,E2 -966.329} C_VEL
LIN {X 0,Y 594.358,Z 136.725,A -85,B 0,C 180,E1 -966.387,E2 -966.387} C_VEL
LIN {X 0,Y 594.391,Z 121.448,A -85,B 0,C 180,E1 -969.224,E2 -969.224} C_VEL
LIN {X 0,Y 594.397,Z 114.441,A -85,B 0,C 180,E1 -970.577,E2 -970.577} C_VEL
LIN {X 0,Y 594.396,Z 114.445,A -85,B 0,C 180,E1 -973.515,E2 -973.515} C_VEL
LIN {X 0,Y 594.375,Z 114.443,A -85,B 0,C 180,E1 -976.321,E2 -976.321} C_VEL
LIN {X 0,Y 594.368,Z 114.444,A -85,B 0,C 180,E1 -979.095,E2 -979.095} C_VEL
LIN {X 0,Y 594.413,Z 114.442,A -85,B 0,C 180,E1 -981.843,E2 -981.843} C_VEL
LIN {X 0,Y 594.382,Z 114.44,A -85,B 0,C 180,E1 -984.572,E2 -984.572} C_VEL
LIN {X 0,Y 594.409,Z 114.445,A -85,B 0,C 180,E1 -987.289,E2 -987.289} C_VEL
LIN {X 0,Y 594.414,Z 114.438,A -85,B 0,C 180,E1 -990,E2 -990} C_VEL
LIN {X 0,Y 594.392,Z 114.441,A -85,B 0,C 180,E1 -992.711,E2 -992.711} C_VEL
LIN {X 0,Y 594.402,Z 114.444,A -85,B 0,C 180,E1 -995.428,E2 -995.428} C_VEL
LIN {X 0,Y 594.381,Z 114.441,A -85,B 0,C 180,E1 -998.157,E2 -998.157} C_VEL
LIN {X 0,Y 594.384,Z 114.451,A -85,B 0,C 180,E1 -1001.071,E2 -1001.071} C_VEL
LIN {X 0,Y 594.381,Z 114.442,A -85,B 0,C 180,E1 -1003.679,E2 -1003.679} C_VEL
LIN {X 0,Y 594.386,Z 114.443,A -85,B 0,C 180,E1 -1006.486,E2 -1006.486} C_VEL
LIN {X 0,Y 594.366,Z 114.445,A -85,B 0,C 180,E1 -1009.334,E2 -1009.334} C_VEL
LIN {X 0,Y 594.363,Z 114.444,A -85,B 0,C 180,E1 -1011.503,E2 -1011.503} C_VEL
LIN {X 0,Y 594.388,Z 114.445,A -85,B 0,C 180,E1 -1014.446,E2 -1014.446} C_VEL
LIN {X 0,Y 594.382,Z 114.451,A -85,B 0,C 180,E1 -1016.699,E2 -1016.699} C_VEL
LIN {X 0,Y 594.38,Z 114.445,A -85,B 0,C 180,E1 -1018.998,E2 -1018.998} C_VEL
LIN {X 0,Y 594.382,Z 114.44,A -85,B 0,C 180,E1 -1021.643,E2 -1021.643} C_VEL
LIN {X 0,Y 594.377,Z 114.45,A -85,B 0,C 180,E1 -1024.58,E2 -1024.58} C_VEL
LIN {X 0,Y 594.388,Z 114.44,A -85,B 0,C 180,E1 -1027.608,E2 -1027.608} C_VEL
LIN {X 0,Y 594.368,Z 114.448,A -85,B 0,C 180,E1 -1030.567,E2 -1030.567} C_VEL
LIN {X 0,Y 594.366,Z 114.442,A -85,B 0,C 180,E1 -1033.299,E2 -1033.299} C_VEL
LIN {X 0,Y 594.367,Z 114.452,A -85,B 0,C 180,E1 -1036.16,E2 -1036.16} C_VEL
LIN {X 0,Y 594.376,Z 114.441,A -85,B 0,C 180,E1 -1039.178,E2 -1039.178} C_VEL
LIN {X 0,Y 594.384,Z 114.451,A -85,B 0,C 180,E1 -1042.059,E2 -1042.059} C_VEL
LIN {X 0,Y 594.35,Z 114.445,A -85,B 0,C 180,E1 -1044.676,E2 -1044.676} C_VEL
LIN {X 0,Y 594.376,Z 114.441,A -85,B 0,C 180,E1 -1047.088,E2 -1047.088} C_VEL
LIN {X 0,Y 594.398,Z 114.445,A -85,B 0,C 180,E1 -1049.669,E2 -1049.669} C_VEL
LIN {X 0,Y 594.372,Z 114.442,A -85,B 0,C 180,E1 -1052.539,E2 -1052.539} C_VEL
LIN {X 0,Y 594.373,Z 114.442,A -85,B 0,C 180,E1 -1054.807,E2 -1054.807} C_VEL
LIN {X 0,Y 594.36,Z 114.447,A -85,B 0,C 180,E1 -1057.265,E2 -1057.265} C_VEL
LIN {X 0,Y 594.373,Z 114.446,A -85,B 0,C 180,E1 -1059.946,E2 -1059.946} C_VEL
LIN {X 0,Y 594.386,Z 114.441,A -85,B 0,C 180,E1 -1062.807,E2 -1062.807} C_VEL
LIN {X 0,Y 594.387,Z 114.444,A -85,B 0,C 180,E1 -1065.826,E2 -1065.826} C_VEL
LIN {X 0,Y 594.384,Z 114.44,A -85,B 0,C 180,E1 -1068.404,E2 -1068.404} C_VEL
LIN {X 0,Y 594.396,Z 114.446,A -85,B 0,C 180,E1 -1071.158,E2 -1071.158} C_VEL
LIN {X 0,Y 594.393,Z 114.44,A -85,B 0,C 180,E1 -1073.891,E2 -1073.891} C_VEL
LIN {X 0,Y 594.373,Z 114.443,A -85,B 0,C 180,E1 -1076.611,E2 -1076.611} C_VEL
LIN {X 0,Y 594.422,Z 114.442,A -85,B 0,C 180,E1 -1079.323,E2 -1079.323} C_VEL
LIN {X 0,Y 594.406,Z 114.437,A -85,B 0,C 180,E1 -1082.033,E2 -1082.033} C_VEL
LIN {X 0,Y 594.385,Z 114.446,A -85,B 0,C 180,E1 -1084.748,E2 -1084.748} C_VEL
LIN {X 0,Y 594.393,Z 114.441,A -85,B 0,C 180,E1 -1087.473,E2 -1087.473} C_VEL
LIN {X 0,Y 594.395,Z 114.44,A -85,B 0,C 180,E1 -1090.216,E2 -1090.216} C_VEL
LIN {X 0,Y 594.364,Z 114.449,A -85,B 0,C 180,E1 -1092.983,E2 -1092.983} C_VEL
LIN {X 0,Y 594.37,Z 114.446,A -85,B 0,C 180,E1 -1095.078,E2 -1095.078} C_VEL
LIN {X 0,Y 594.388,Z 114.442,A -85,B 0,C 180,E1 -1097.194,E2 -1097.194} C_VEL
LIN {X 0,Y 594.373,Z 114.444,A -85,B 0,C 180,E1 -1100.054,E2 -1100.054} C_VEL
LIN {X 0,Y 594.363,Z 114.446,A -85,B 0,C 180,E1 -1102.968,E2 -1102.968} C_VEL
LIN {X 0,Y 594.374,Z 114.442,A -85,B 0,C 180,E1 -1105.193,E2 -1105.193} C_VEL
LIN {X 0,Y 594.385,Z 114.44,A -85,B 0,C 180,E1 -1107.527,E2 -1107.527} C_VEL
LIN {X 0,Y 594.386,Z 114.45,A -85,B 0,C 180,E1 -1110.329,E2 -1110.329} C_VEL
LIN {X 0,Y 594.379,Z 114.442,A -85,B 0,C 180,E1 -1112.95,E2 -1112.95} C_VEL
LIN {X 0,Y 594.349,Z 114.445,A -85,B 0,C 180,E1 -1115.409,E2 -1115.409} C_VEL
LIN {X 0,Y 594.39,Z 114.446,A -85,B 0,C 180,E1 -1117.941,E2 -1117.941} C_VEL
LIN {X 0,Y 594.379,Z 114.441,A -85,B 0,C 180,E1 -1120.823,E2 -1120.823} C_VEL
LIN {X 0,Y 594.367,Z 114.443,A -85,B 0,C 180,E1 -1123.3,E2 -1123.3} C_VEL
LIN {X 0,Y 594.369,Z 114.449,A -85,B 0,C 180,E1 -1126.161,E2 -1126.161} C_VEL
LIN {X 0,Y 594.382,Z 114.442,A -85,B 0,C 180,E1 -1128.537,E2 -1128.537} C_VEL
LIN {X 0,Y 594.389,Z 114.442,A -85,B 0,C 180,E1 -1131.295,E2 -1131.295} C_VEL
LIN {X 0,Y 594.353,Z 114.455,A -85,B 0,C 180,E1 -1133.756,E2 -1133.756} C_VEL
LIN {X 0,Y 594.377,Z 114.443,A -85,B 0,C 180,E1 -1136.239,E2 -1136.239} C_VEL
LIN {X 0,Y 594.371,Z 114.442,A -85,B 0,C 180,E1 -1138.65,E2 -1138.65} C_VEL
LIN {X 0,Y 594.386,Z 114.443,A -85,B 0,C 180,E1 -1141.042,E2 -1141.042} C_VEL
LIN {X 0,Y 594.385,Z 114.444,A -85,B 0,C 180,E1 -1143.978,E2 -1143.978} C_VEL
LIN {X 0,Y 594.396,Z 114.515,A -85,B 0,C 180,E1 -1146.204,E2 -1146.204} C_VEL
LIN {X 0,Y 594.863,Z 118.015,A -85,B 0,C 180,E1 -1146.685,E2 -1146.685} C_VEL
LIN {X 0,Y 594.693,Z 139.851,A -85,B 0,C 180,E1 -1149.597,E2 -1149.597} C_VEL
LIN {X 0,Y 594.579,Z 163.051,A -85,B 0,C 180,E1 -1152.635,E2 -1152.635} C_VEL
LIN {X 0,Y 594.465,Z 183.522,A -85,B 0,C 180,E1 -1155.275,E2 -1155.275} C_VEL
LIN {X 0,Y 594.422,Z 194.355,A -85,B 0,C 180,E1 -1156.66,E2 -1156.66} C_VEL
LIN {X 0,Y 594.75,Z 200.513,A -85,B 0,C 180,E1 -1156.743,E2 -1156.743} C_VEL
LIN {X 0,Y 594.665,Z 302.949,A -85,B 0,C 180,E1 -1157.999,E2 -1157.999} C_VEL
LIN {X 0,Y 594.601,Z 316.22,A -85,B 0,C 180,E1 -1158.3,E2 -1158.3} C_VEL
LIN {X 0,Y 594.59,Z 329.277,A -85,B 0,C 180,E1 -1158.746,E2 -1158.746} C_VEL
LIN {X 0,Y 594.536,Z 340.632,A -85,B 0,C 180,E1 -1159.27,E2 -1159.27} C_VEL
LIN {X 0,Y 594.477,Z 352.202,A -85,B 0,C 180,E1 -1159.958,E2 -1159.958} C_VEL
LIN {X 0,Y 594.414,Z 362.598,A -85,B 0,C 180,E1 -1160.73,E2 -1160.73} C_VEL
LIN {X 0,Y 594.383,Z 371.112,A -85,B 0,C 180,E1 -1161.501,E2 -1161.501} C_VEL
LIN {X 0,Y 594.347,Z 378.961,A -85,B 0,C 180,E1 -1162.355,E2 -1162.355} C_VEL
LIN {X 0,Y 594.282,Z 386.814,A -85,B 0,C 180,E1 -1163.408,E2 -1163.408} C_VEL
LIN {X 0,Y 594.289,Z 393.68,A -85,B 0,C 180,E1 -1164.571,E2 -1164.571} C_VEL
LIN {X 0,Y 594.27,Z 398.371,A -85,B 0,C 180,E1 -1165.591,E2 -1165.591} C_VEL
LIN {X 0,Y 594.267,Z 401.956,A -85,B 0,C 180,E1 -1166.61,E2 -1166.61} C_VEL
LIN {X 0,Y 594.226,Z 403.809,A -85,B 0,C 180,E1 -1167.288,E2 -1167.288} C_VEL
LIN {X 0,Y 594.242,Z 405.201,A -85,B 0,C 180,E1 -1167.967,E2 -1167.967} C_VEL
LIN {X 0,Y 594.239,Z 406.784,A -85,B 0,C 180,E1 -1169.322,E2 -1169.322} C_VEL
LIN {X 0,Y 594.236,Z 407,A -85,B 0,C 180,E1 -1170,E2 -1170} C_VEL
LIN {X 0,Y 594.247,Z 406.185,A -85,B 0,C 180,E1 -1171.355,E2 -1171.355} C_VEL
LIN {X 0,Y 594.242,Z 405.201,A -85,B 0,C 180,E1 -1172.033,E2 -1172.033} C_VEL
LIN {X 0,Y 594.226,Z 403.81,A -85,B 0,C 180,E1 -1172.712,E2 -1172.712} C_VEL
LIN {X 0,Y 594.289,Z 400.896,A -85,B 0,C 180,E1 -1173.729,E2 -1173.729} C_VEL
LIN {X 0,Y 594.241,Z 396.95,A -85,B 0,C 180,E1 -1174.749,E2 -1174.749} C_VEL
LIN {X 0,Y 594.305,Z 390.878,A -85,B 0,C 180,E1 -1175.939,E2 -1175.939} C_VEL
LIN {X 0,Y 594.308,Z 384.237,A -85,B 0,C 180,E1 -1176.962,E2 -1176.962} C_VEL
LIN {X 0,Y 594.359,Z 375.991,A -85,B 0,C 180,E1 -1177.986,E2 -1177.986} C_VEL
LIN {X 0,Y 594.382,Z 367.538,A -85,B 0,C 180,E1 -1178.842,E2 -1178.842} C_VEL
LIN {X 0,Y 594.432,Z 357.096,A -85,B 0,C 180,E1 -1179.699,E2 -1179.699} C_VEL
LIN {X 0,Y 594.481,Z 346.76,A -85,B 0,C 180,E1 -1180.386,E2 -1180.386} C_VEL
LIN {X 0,Y 594.558,Z 335.725,A -85,B 0,C 180,E1 -1180.973,E2 -1180.973} C_VEL
LIN {X 0,Y 594.579,Z 323.714,A -85,B 0,C 180,E1 -1181.464,E2 -1181.464} C_VEL
LIN {X 0,Y 594.647,Z 310.355,A -85,B 0,C 180,E1 -1181.85,E2 -1181.85} C_VEL
LIN {X 0,Y 594.697,Z 297.092,A -85,B 0,C 180,E1 -1182.087,E2 -1182.087} C_VEL
LIN {X 0,Y 594.622,Z 195.822,A -85,B 0,C 180,E1 -1183.317,E2 -1183.317} C_VEL
LIN {X 0,Y 594.429,Z 194.27,A -85,B 0,C 180,E1 -1183.351,E2 -1183.351} C_VEL
LIN {X 0,Y 594.529,Z 171.24,A -85,B 0,C 180,E1 -1186.305,E2 -1186.305} C_VEL
LIN {X 0,Y 594.613,Z 153.499,A -85,B 0,C 180,E1 -1188.61,E2 -1188.61} C_VEL
LIN {X 0,Y 594.747,Z 132.811,A -85,B 0,C 180,E1 -1191.336,E2 -1191.336} C_VEL
LIN {X 0,Y 594.819,Z 116.632,A -85,B 0,C 180,E1 -1193.501,E2 -1193.501} C_VEL
LIN {X 0,Y 594.391,Z 114.445,A -85,B 0,C 180,E1 -1193.819,E2 -1193.819} C_VEL
LIN {X 0,Y 594.385,Z 114.447,A -85,B 0,C 180,E1 -1196.699,E2 -1196.699} C_VEL
LIN {X 0,Y 594.383,Z 114.443,A -85,B 0,C 180,E1 -1198.998,E2 -1198.998} C_VEL
LIN {X 0,Y 594.379,Z 114.442,A -85,B 0,C 180,E1 -1201.642,E2 -1201.642} C_VEL
LIN {X 0,Y 594.379,Z 114.447,A -85,B 0,C 180,E1 -1204.58,E2 -1204.58} C_VEL
LIN {X 0,Y 594.392,Z 114.441,A -85,B 0,C 180,E1 -1207.608,E2 -1207.608} C_VEL
LIN {X 0,Y 594.372,Z 114.446,A -85,B 0,C 180,E1 -1210.566,E2 -1210.566} C_VEL
LIN {X 0,Y 594.367,Z 114.443,A -85,B 0,C 180,E1 -1213.299,E2 -1213.299} C_VEL
LIN {X 0,Y 594.369,Z 114.451,A -85,B 0,C 180,E1 -1216.16,E2 -1216.16} C_VEL
LIN {X 0,Y 594.379,Z 114.441,A -85,B 0,C 180,E1 -1219.177,E2 -1219.177} C_VEL
LIN {X 0,Y 594.387,Z 114.448,A -85,B 0,C 180,E1 -1222.059,E2 -1222.059} C_VEL
LIN {X 0,Y 594.349,Z 114.445,A -85,B 0,C 180,E1 -1224.676,E2 -1224.676} C_VEL
LIN {X 0,Y 594.378,Z 114.442,A -85,B 0,C 180,E1 -1227.088,E2 -1227.088} C_VEL
LIN {X 0,Y 594.386,Z 114.449,A -85,B 0,C 180,E1 -1229.671,E2 -1229.671} C_VEL
LIN {X 0,Y 594.373,Z 114.442,A -85,B 0,C 180,E1 -1232.539,E2 -1232.539} C_VEL
LIN {X 0,Y 594.374,Z 114.441,A -85,B 0,C 180,E1 -1234.807,E2 -1234.807} C_VEL
LIN {X 0,Y 594.361,Z 114.448,A -85,B 0,C 180,E1 -1237.265,E2 -1237.265} C_VEL
LIN {X 0,Y 594.374,Z 114.444,A -85,B 0,C 180,E1 -1239.946,E2 -1239.946} C_VEL
LIN {X 0,Y 594.387,Z 114.441,A -85,B 0,C 180,E1 -1242.806,E2 -1242.806} C_VEL
LIN {X 0,Y 594.387,Z 114.443,A -85,B 0,C 180,E1 -1245.826,E2 -1245.826} C_VEL
LIN {X 0,Y 594.391,Z 114.439,A -85,B 0,C 180,E1 -1248.404,E2 -1248.404} C_VEL
LIN {X 0,Y 594.395,Z 114.448,A -85,B 0,C 180,E1 -1251.158,E2 -1251.158} C_VEL
LIN {X 0,Y 594.392,Z 114.44,A -85,B 0,C 180,E1 -1253.891,E2 -1253.891} C_VEL
LIN {X 0,Y 594.374,Z 114.443,A -85,B 0,C 180,E1 -1256.61,E2 -1256.61} C_VEL
LIN {X 0,Y 594.42,Z 114.441,A -85,B 0,C 180,E1 -1259.322,E2 -1259.322} C_VEL
LIN {X 0,Y 594.406,Z 114.437,A -85,B 0,C 180,E1 -1262.033,E2 -1262.033} C_VEL
LIN {X 0,Y 594.386,Z 114.447,A -85,B 0,C 180,E1 -1264.748,E2 -1264.748} C_VEL
LIN {X 0,Y 594.392,Z 114.441,A -85,B 0,C 180,E1 -1267.473,E2 -1267.473} C_VEL
LIN {X 0,Y 594.395,Z 114.44,A -85,B 0,C 180,E1 -1270.216,E2 -1270.216} C_VEL
LIN {X 0,Y 594.364,Z 114.449,A -85,B 0,C 180,E1 -1272.983,E2 -1272.983} C_VEL
LIN {X 0,Y 594.358,Z 114.445,A -85,B 0,C 180,E1 -1275.323,E2 -1275.323} C_VEL
LIN {X 0,Y 593.683,Z 114.529,A -85,B 0,C 180,E1 -1275.888,E2 -1275.888} C_VEL
LIN {X 0,Y 590.817,Z 114.893,A -85,B 0,C 180,E1 -1276.807,E2 -1276.807} C_VEL
LIN {X 0,Y 588.407,Z 115.19,A -85,B 0,C 180,E1 -1277.545,E2 -1277.545} C_VEL
LIN {X 0,Y 587.385,Z 115.315,A -85,B 0,C 180,E1 -1278.115,E2 -1278.115} C_VEL
LIN {X 0,Y 587.309,Z 115.324,A -85,B 0,C 180,E1 -1278.308,E2 -1278.308} C_VEL
LIN {X 0,Y 587.328,Z 115.323,A -85,B 0,C 180,E1 -1281.038,E2 -1281.038} C_VEL
LIN {X 0,Y 587.319,Z 115.322,A -85,B 0,C 180,E1 -1283.259,E2 -1283.259} C_VEL
LIN {X 0,Y 587.333,Z 115.319,A -85,B 0,C 180,E1 -1285.517,E2 -1285.517} C_VEL
LIN {X 0,Y 587.347,Z 115.319,A -85,B 0,C 180,E1 -1287.818,E2 -1287.818} C_VEL
LIN {X 0,Y 587.339,Z 115.326,A -85,B 0,C 180,E1 -1290.511,E2 -1290.511} C_VEL
LIN {X 0,Y 587.338,Z 115.319,A -85,B 0,C 180,E1 -1293.112,E2 -1293.112} C_VEL
LIN {X 0,Y 587.361,Z 115.399,A -85,B 0,C 180,E1 -1295.518,E2 -1295.518} C_VEL
LIN {X 0,Y 587.352,Z 127.664,A -85,B 0,C 180,E1 -1297.841,E2 -1297.841} C_VEL
LIN {X 0,Y 587.325,Z 136.917,A -85,B 0,C 180,E1 -1299.573,E2 -1299.573} C_VEL
LIN {X 0,Y 587.829,Z 142.251,A -85,B 0,C 180,E1 -1299.651,E2 -1299.651} C_VEL
LIN {X 0,Y 587.714,Z 243.57,A -85,B 0,C 180,E1 -1300.912,E2 -1300.912} C_VEL
LIN {X 0,Y 587.652,Z 256.814,A -85,B 0,C 180,E1 -1301.222,E2 -1301.222} C_VEL
LIN {X 0,Y 587.596,Z 269.111,A -85,B 0,C 180,E1 -1301.648,E2 -1301.648} C_VEL
LIN {X 0,Y 587.5,Z 281.649,A -85,B 0,C 180,E1 -1302.241,E2 -1302.241} C_VEL
LIN {X 0,Y 587.485,Z 292.103,A -85,B 0,C 180,E1 -1302.875,E2 -1302.875} C_VEL
LIN {X 0,Y 587.399,Z 303.345,A -85,B 0,C 180,E1 -1303.724,E2 -1303.724} C_VEL
LIN {X 0,Y 587.315,Z 312.817,A -85,B 0,C 180,E1 -1304.619,E2 -1304.619} C_VEL
LIN {X 0,Y 587.276,Z 320.629,A -85,B 0,C 180,E1 -1305.518,E2 -1305.518} C_VEL
LIN {X 0,Y 587.229,Z 327.592,A -85,B 0,C 180,E1 -1306.494,E2 -1306.494} C_VEL
LIN {X 0,Y 587.218,Z 334.376,A -85,B 0,C 180,E1 -1307.685,E2 -1307.685} C_VEL
LIN {X 0,Y 587.138,Z 339.752,A -85,B 0,C 180,E1 -1308.947,E2 -1308.947} C_VEL
LIN {X 0,Y 587.157,Z 343.039,A -85,B 0,C 180,E1 -1310,E2 -1310} C_VEL
LIN {X 0,Y 587.113,Z 345.36,A -85,B 0,C 180,E1 -1311.085,E2 -1311.085} C_VEL
LIN {X 0,Y 587.14,Z 346.797,A -85,B 0,C 180,E1 -1312.377,E2 -1312.377} C_VEL
LIN {X 0,Y 587.123,Z 346.943,A -85,B 0,C 180,E1 -1313.322,E2 -1313.322} C_VEL
LIN {X 0,Y 587.132,Z 346.107,A -85,B 0,C 180,E1 -1314.485,E2 -1314.485} C_VEL
LIN {X 0,Y 587.143,Z 343.864,A -85,B 0,C 180,E1 -1315.766,E2 -1315.766} C_VEL
LIN {X 0,Y 587.153,Z 340.566,A -85,B 0,C 180,E1 -1316.916,E2 -1316.916} C_VEL
LIN {X 0,Y 587.197,Z 335.4,A -85,B 0,C 180,E1 -1318.188,E2 -1318.188} C_VEL
LIN {X 0,Y 587.239,Z 329.467,A -85,B 0,C 180,E1 -1319.297,E2 -1319.297} C_VEL
LIN {X 0,Y 587.251,Z 321.832,A -85,B 0,C 180,E1 -1320.419,E2 -1320.419} C_VEL
LIN {X 0,Y 587.308,Z 313.462,A -85,B 0,C 180,E1 -1321.402,E2 -1321.402} C_VEL
LIN {X 0,Y 587.374,Z 304.076,A -85,B 0,C 180,E1 -1322.303,E2 -1322.303} C_VEL
LIN {X 0,Y 587.466,Z 293.017,A -85,B 0,C 180,E1 -1323.153,E2 -1323.153} C_VEL
LIN {X 0,Y 587.513,Z 281.333,A -85,B 0,C 180,E1 -1323.866,E2 -1323.866} C_VEL
LIN {X 0,Y 587.596,Z 268.941,A -85,B 0,C 180,E1 -1324.448,E2 -1324.448} C_VEL
LIN {X 0,Y 587.674,Z 256.434,A -85,B 0,C 180,E1 -1324.878,E2 -1324.878} C_VEL
LIN {X 0,Y 587.747,Z 242.985,A -85,B 0,C 180,E1 -1325.189,E2 -1325.189} C_VEL
LIN {X 0,Y 587.716,Z 139.331,A -85,B 0,C 180,E1 -1326.478,E2 -1326.478} C_VEL
LIN {X 0,Y 587.324,Z 136.825,A -85,B 0,C 180,E1 -1326.532,E2 -1326.532} C_VEL
LIN {X 0,Y 587.372,Z 121.933,A -85,B 0,C 180,E1 -1329.331,E2 -1329.331} C_VEL
LIN {X 0,Y 587.36,Z 115.318,A -85,B 0,C 180,E1 -1330.623,E2 -1330.623} C_VEL
LIN {X 0,Y 587.329,Z 115.323,A -85,B 0,C 180,E1 -1333.311,E2 -1333.311} C_VEL
LIN {X 0,Y 587.355,Z 115.319,A -85,B 0,C 180,E1 -1336.154,E2 -1336.154} C_VEL
LIN {X 0,Y 587.337,Z 115.319,A -85,B 0,C 180,E1 -1338.962,E2 -1338.962} C_VEL
LIN {X 0,Y 587.365,Z 115.321,A -85,B 0,C 180,E1 -1341.745,E2 -1341.745} C_VEL
LIN {X 0,Y 587.351,Z 115.316,A -85,B 0,C 180,E1 -1344.507,E2 -1344.507} C_VEL
LIN {X 0,Y 587.374,Z 115.321,A -85,B 0,C 180,E1 -1347.257,E2 -1347.257} C_VEL
LIN {X 0,Y 587.383,Z 115.313,A -85,B 0,C 180,E1 -1350,E2 -1350} C_VEL
LIN {X 0,Y 587.36,Z 115.317,A -85,B 0,C 180,E1 -1352.743,E2 -1352.743} C_VEL
LIN {X 0,Y 587.367,Z 115.32,A -85,B 0,C 180,E1 -1355.493,E2 -1355.493} C_VEL
LIN {X 0,Y 587.34,Z 115.318,A -85,B 0,C 180,E1 -1358.256,E2 -1358.256} C_VEL
LIN {X 0,Y 587.349,Z 115.326,A -85,B 0,C 180,E1 -1361.134,E2 -1361.134} C_VEL
LIN {X 0,Y 587.365,Z 115.315,A -85,B 0,C 180,E1 -1364.26,E2 -1364.26} C_VEL
LIN {X 0,Y 587.34,Z 115.32,A -85,B 0,C 180,E1 -1367.406,E2 -1367.406} C_VEL
LIN {X 0,Y 587.311,Z 115.322,A -85,B 0,C 180,E1 -1369.576,E2 -1369.576} C_VEL
LIN {X 0,Y 587.337,Z 115.324,A -85,B 0,C 180,E1 -1372.514,E2 -1372.514} C_VEL
LIN {X 0,Y 587.33,Z 115.319,A -85,B 0,C 180,E1 -1375.517,E2 -1375.517} C_VEL
LIN {X 0,Y 587.346,Z 115.317,A -85,B 0,C 180,E1 -1377.818,E2 -1377.818} C_VEL
LIN {X 0,Y 587.328,Z 115.328,A -85,B 0,C 180,E1 -1380.508,E2 -1380.508} C_VEL
LIN {X 0,Y 587.336,Z 115.32,A -85,B 0,C 180,E1 -1383.111,E2 -1383.111} C_VEL
LIN {X 0,Y 587.289,Z 115.326,A -85,B 0,C 180,E1 -1385.9,E2 -1385.9} C_VEL
LIN {X 0,Y 587.327,Z 115.328,A -85,B 0,C 180,E1 -1388.479,E2 -1388.479} C_VEL
LIN {X 0,Y 587.334,Z 115.319,A -85,B 0,C 180,E1 -1391.157,E2 -1391.157} C_VEL
LIN {X 0,Y 587.325,Z 115.327,A -85,B 0,C 180,E1 -1394.113,E2 -1394.113} C_VEL
LIN {X 0,Y 587.312,Z 115.321,A -85,B 0,C 180,E1 -1396.993,E2 -1396.993} C_VEL
LIN {X 0,Y 587.316,Z 115.325,A -85,B 0,C 180,E1 -1399.746,E2 -1399.746} C_VEL
LIN {X 0,Y 587.344,Z 115.322,A -85,B 0,C 180,E1 -1402.392,E2 -1402.392} C_VEL
LIN {X 0,Y 587.345,Z 115.322,A -85,B 0,C 180,E1 -1405.652,E2 -1405.652} C_VEL
LIN {X 0,Y 587.343,Z 115.322,A -85,B 0,C 180,E1 -1408.231,E2 -1408.231} C_VEL
LIN {X 0,Y 587.348,Z 115.317,A -85,B 0,C 180,E1 -1410.866,E2 -1410.866} C_VEL
LIN {X 0,Y 587.358,Z 115.325,A -85,B 0,C 180,E1 -1413.819,E2 -1413.819} C_VEL
LIN {X 0,Y 587.329,Z 115.324,A -85,B 0,C 180,E1 -1415.993,E2 -1415.993} C_VEL
LIN {X 0,Y 587.322,Z 115.322,A -85,B 0,C 180,E1 -1418.226,E2 -1418.226} C_VEL
LIN {X 0,Y 587.347,Z 115.32,A -85,B 0,C 180,E1 -1421.151,E2 -1421.151} C_VEL
LIN {X 0,Y 587.323,Z 115.322,A -85,B 0,C 180,E1 -1424.025,E2 -1424.025} C_VEL
LIN {X 0,Y 587.356,Z 115.317,A -85,B 0,C 180,E1 -1426.154,E2 -1426.154} C_VEL
LIN {X 0,Y 587.34,Z 115.321,A -85,B 0,C 180,E1 -1428.963,E2 -1428.963} C_VEL
LIN {X 0,Y 587.37,Z 115.317,A -85,B 0,C 180,E1 -1431.745,E2 -1431.745} C_VEL
LIN {X 0,Y 587.358,Z 115.316,A -85,B 0,C 180,E1 -1434.507,E2 -1434.507} C_VEL
LIN {X 0,Y 587.37,Z 115.323,A -85,B 0,C 180,E1 -1437.257,E2 -1437.257} C_VEL
LIN {X 0,Y 587.383,Z 115.312,A -85,B 0,C 180,E1 -1440,E2 -1440} C_VEL
LIN {X 0,Y 587.368,Z 115.319,A -85,B 0,C 180,E1 -1442.743,E2 -1442.743} C_VEL
LIN {X 0,Y 587.363,Z 115.317,A -85,B 0,C 180,E1 -1445.493,E2 -1445.493} C_VEL
LIN {X 0,Y 587.363,Z 115.316,A -85,B 0,C 180,E1 -1448.255,E2 -1448.255} C_VEL
LIN {X 0,Y 587.347,Z 115.322,A -85,B 0,C 180,E1 -1451.134,E2 -1451.134} C_VEL
LIN {X 0,Y 587.364,Z 115.317,A -85,B 0,C 180,E1 -1454.261,E2 -1454.261} C_VEL
LIN {X 0,Y 587.348,Z 115.317,A -85,B 0,C 180,E1 -1457.406,E2 -1457.406} C_VEL
LIN {X 0,Y 587.329,Z 115.324,A -85,B 0,C 180,E1 -1460.305,E2 -1460.305} C_VEL
LIN {X 0,Y 587.32,Z 115.321,A -85,B 0,C 180,E1 -1463.259,E2 -1463.259} C_VEL
LIN {X 0,Y 587.334,Z 115.318,A -85,B 0,C 180,E1 -1465.517,E2 -1465.517} C_VEL
LIN {X 0,Y 587.347,Z 115.319,A -85,B 0,C 180,E1 -1467.818,E2 -1467.818} C_VEL
LIN {X 0,Y 587.338,Z 115.325,A -85,B 0,C 180,E1 -1470.511,E2 -1470.511} C_VEL
LIN {X 0,Y 587.335,Z 115.318,A -85,B 0,C 180,E1 -1473.397,E2 -1473.397} C_VEL
LIN {X 0,Y 587.291,Z 115.329,A -85,B 0,C 180,E1 -1475.9,E2 -1475.9} C_VEL
LIN {X 0,Y 587.335,Z 115.323,A -85,B 0,C 180,E1 -1478.479,E2 -1478.479} C_VEL
LIN {X 0,Y 587.337,Z 115.318,A -85,B 0,C 180,E1 -1481.157,E2 -1481.157} C_VEL
LIN {X 0,Y 587.328,Z 115.327,A -85,B 0,C 180,E1 -1484.114,E2 -1484.114} C_VEL
LIN {X 0,Y 587.316,Z 115.321,A -85,B 0,C 180,E1 -1486.994,E2 -1486.994} C_VEL
LIN {X 0,Y 587.319,Z 115.328,A -85,B 0,C 180,E1 -1489.746,E2 -1489.746} C_VEL
LIN {X 0,Y 587.347,Z 115.318,A -85,B 0,C 180,E1 -1492.393,E2 -1492.393} C_VEL
LIN {X 0,Y 587.361,Z 115.324,A -85,B 0,C 180,E1 -1495.78,E2 -1495.78} C_VEL
LIN {X 0,Y 587.343,Z 115.319,A -85,B 0,C 180,E1 -1498.231,E2 -1498.231} C_VEL
LIN {X 0,Y 587.352,Z 115.318,A -85,B 0,C 180,E1 -1500.867,E2 -1500.867} C_VEL
LIN {X 0,Y 587.36,Z 115.322,A -85,B 0,C 180,E1 -1503.819,E2 -1503.819} C_VEL
LIN {X 0,Y 587.384,Z 115.409,A -85,B 0,C 180,E1 -1506.066,E2 -1506.066} C_VEL
LIN {X 0,Y 587.926,Z 119.104,A -85,B 0,C 180,E1 -1506.58,E2 -1506.58} C_VEL
LIN {X 0,Y 587.771,Z 138.486,A -85,B 0,C 180,E1 -1509.162,E2 -1509.162} C_VEL
LIN {X 0,Y 587.678,Z 158.957,A -85,B 0,C 180,E1 -1511.885,E2 -1511.885} C_VEL
LIN {X 0,Y 587.5,Z 180.793,A -85,B 0,C 180,E1 -1514.741,E2 -1514.741} C_VEL
LIN {X 0,Y 587.386,Z 194.355,A -85,B 0,C 180,E1 -1516.497,E2 -1516.497} C_VEL
LIN {X 0,Y 587.862,Z 200.513,A -85,B 0,C 180,E1 -1516.585,E2 -1516.585} C_VEL
LIN {X 0,Y 587.726,Z 302.949,A -85,B 0,C 180,E1 -1517.855,E2 -1517.855} C_VEL
LIN {X 0,Y 587.655,Z 316.221,A -85,B 0,C 180,E1 -1518.16,E2 -1518.16} C_VEL
LIN {X 0,Y 587.613,Z 328.646,A -85,B 0,C 180,E1 -1518.586,E2 -1518.586} C_VEL
LIN {X 0,Y 587.557,Z 340.63,A -85,B 0,C 180,E1 -1519.141,E2 -1519.141} C_VEL
LIN {X 0,Y 587.464,Z 352.204,A -85,B 0,C 180,E1 -1519.836,E2 -1519.836} C_VEL
LIN {X 0,Y 587.394,Z 362.599,A -85,B 0,C 180,E1 -1520.618,E2 -1520.618} C_VEL
LIN {X 0,Y 587.322,Z 371.113,A -85,B 0,C 180,E1 -1521.398,E2 -1521.398} C_VEL
LIN {X 0,Y 587.274,Z 378.961,A -85,B 0,C 180,E1 -1522.263,E2 -1522.263} C_VEL
LIN {X 0,Y 587.23,Z 385.469,A -85,B 0,C 180,E1 -1523.126,E2 -1523.126} C_VEL
LIN {X 0,Y 587.237,Z 391.867,A -85,B 0,C 180,E1 -1524.161,E2 -1524.161} C_VEL
LIN {X 0,Y 587.147,Z 396.95,A -85,B 0,C 180,E1 -1525.194,E2 -1525.194} C_VEL
LIN {X 0,Y 587.213,Z 400.895,A -85,B 0,C 180,E1 -1526.226,E2 -1526.226} C_VEL
LIN {X 0,Y 587.132,Z 403.808,A -85,B 0,C 180,E1 -1527.256,E2 -1527.256} C_VEL
LIN {X 0,Y 587.141,Z 405.199,A -85,B 0,C 180,E1 -1527.942,E2 -1527.942} C_VEL
LIN {X 0,Y 587.14,Z 406.785,A -85,B 0,C 180,E1 -1529.314,E2 -1529.314} C_VEL
LIN {X 0,Y 587.137,Z 407,A -85,B 0,C 180,E1 -1530,E2 -1530} C_VEL
LIN {X 0,Y 587.147,Z 406.186,A -85,B 0,C 180,E1 -1531.372,E2 -1531.372} C_VEL
LIN {X 0,Y 587.141,Z 405.2,A -85,B 0,C 180,E1 -1532.058,E2 -1532.058} C_VEL
LIN {X 0,Y 587.132,Z 403.81,A -85,B 0,C 180,E1 -1532.744,E2 -1532.744} C_VEL
LIN {X 0,Y 587.213,Z 400.896,A -85,B 0,C 180,E1 -1533.774,E2 -1533.774} C_VEL
LIN {X 0,Y 587.147,Z 396.949,A -85,B 0,C 180,E1 -1534.806,E2 -1534.806} C_VEL
LIN {X 0,Y 587.218,Z 390.878,A -85,B 0,C 180,E1 -1536.011,E2 -1536.011} C_VEL
LIN {X 0,Y 587.245,Z 384.238,A -85,B 0,C 180,E1 -1537.046,E2 -1537.046} C_VEL
LIN {X 0,Y 587.299,Z 375.991,A -85,B 0,C 180,E1 -1538.083,E2 -1538.083} C_VEL
LIN {X 0,Y 587.343,Z 367.539,A -85,B 0,C 180,E1 -1538.949,E2 -1538.949} C_VEL
LIN {X 0,Y 587.419,Z 357.098,A -85,B 0,C 180,E1 -1539.816,E2 -1539.816} C_VEL
LIN {X 0,Y 587.497,Z 346.758,A -85,B 0,C 180,E1 -1540.511,E2 -1540.511} C_VEL
LIN {X 0,Y 587.561,Z 334.819,A -85,B 0,C 180,E1 -1541.149,E2 -1541.149} C_VEL
LIN {X 0,Y 587.629,Z 322.602,A -85,B 0,C 180,E1 -1541.639,E2 -1541.639} C_VEL
LIN {X 0,Y 587.703,Z 309.439,A -85,B 0,C 180,E1 -1542.014,E2 -1542.014} C_VEL
LIN {X 0,Y 587.768,Z 297.092,A -85,B 0,C 180,E1 -1542.232,E2 -1542.232} C_VEL
LIN {X 0,Y 587.714,Z 196.493,A -85,B 0,C 180,E1 -1543.468,E2 -1543.468} C_VEL
LIN {X 0,Y 587.394,Z 194.27,A -85,B 0,C 180,E1 -1543.514,E2 -1543.514} C_VEL
LIN {X 0,Y 587.551,Z 172.605,A -85,B 0,C 180,E1 -1546.325,E2 -1546.325} C_VEL
LIN {X 0,Y 587.641,Z 153.499,A -85,B 0,C 180,E1 -1548.839,E2 -1548.839} C_VEL
LIN {X 0,Y 587.833,Z 134.335,A -85,B 0,C 180,E1 -1551.394,E2 -1551.394} C_VEL
LIN {X 0,Y 587.925,Z 119.005,A -85,B 0,C 180,E1 -1553.42,E2 -1553.42} C_VEL
LIN {X 0,Y 587.37,Z 115.322,A -85,B 0,C 180,E1 -1553.958,E2 -1553.958} C_VEL
LIN {X 0,Y 587.331,Z 115.322,A -85,B 0,C 180,E1 -1557.046,E2 -1557.046} C_VEL
LIN {X 0,Y 587.348,Z 115.318,A -85,B 0,C 180,E1 -1559.379,E2 -1559.379} C_VEL
LIN {X 0,Y 587.347,Z 115.32,A -85,B 0,C 180,E1 -1561.835,E2 -1561.835} C_VEL
LIN {X 0,Y 587.348,Z 115.327,A -85,B 0,C 180,E1 -1564.347,E2 -1564.347} C_VEL
LIN {X 0,Y 587.347,Z 115.319,A -85,B 0,C 180,E1 -1567.607,E2 -1567.607} C_VEL
LIN {X 0,Y 587.319,Z 115.33,A -85,B 0,C 180,E1 -1570.254,E2 -1570.254} C_VEL
LIN {X 0,Y 587.315,Z 115.321,A -85,B 0,C 180,E1 -1573.006,E2 -1573.006} C_VEL
LIN {X 0,Y 587.327,Z 115.327,A -85,B 0,C 180,E1 -1575.886,E2 -1575.886} C_VEL
LIN {X 0,Y 587.337,Z 115.318,A -85,B 0,C 180,E1 -1578.843,E2 -1578.843} C_VEL
LIN {X 0,Y 587.333,Z 115.322,A -85,B 0,C 180,E1 -1581.521,E2 -1581.521} C_VEL
LIN {X 0,Y 587.29,Z 115.33,A -85,B 0,C 180,E1 -1584.1,E2 -1584.1} C_VEL
LIN {X 0,Y 587.334,Z 115.319,A -85,B 0,C 180,E1 -1586.603,E2 -1586.603} C_VEL
LIN {X 0,Y 587.338,Z 115.324,A -85,B 0,C 180,E1 -1589.489,E2 -1589.489} C_VEL
LIN {X 0,Y 587.35,Z 115.318,A -85,B 0,C 180,E1 -1592.307,E2 -1592.307} C_VEL
LIN {X 0,Y 587.334,Z 115.318,A -85,B 0,C 180,E1 -1594.483,E2 -1594.483} C_VEL
LIN {X 0,Y 587.338,Z 115.327,A -85,B 0,C 180,E1 -1597.486,E2 -1597.486} C_VEL
LIN {X 0,Y 587.342,Z 115.317,A -85,B 0,C 180,E1 -1600.425,E2 -1600.425} C_VEL
LIN {X 0,Y 587.35,Z 115.324,A -85,B 0,C 180,E1 -1603.311,E2 -1603.311} C_VEL
LIN {X 0,Y 587.356,Z 115.316,A -85,B 0,C 180,E1 -1606.154,E2 -1606.154} C_VEL
LIN {X 0,Y 587.342,Z 115.322,A -85,B 0,C 180,E1 -1608.962,E2 -1608.962} C_VEL
LIN {X 0,Y 587.369,Z 115.316,A -85,B 0,C 180,E1 -1611.745,E2 -1611.745} C_VEL
LIN {X 0,Y 587.359,Z 115.316,A -85,B 0,C 180,E1 -1614.507,E2 -1614.507} C_VEL
LIN {X 0,Y 587.371,Z 115.322,A -85,B 0,C 180,E1 -1617.257,E2 -1617.257} C_VEL
LIN {X 0,Y 587.383,Z 115.312,A -85,B 0,C 180,E1 -1620,E2 -1620} C_VEL
LIN {X 0,Y 587.368,Z 115.32,A -85,B 0,C 180,E1 -1622.743,E2 -1622.743} C_VEL
LIN {X 0,Y 587.362,Z 115.317,A -85,B 0,C 180,E1 -1625.493,E2 -1625.493} C_VEL
LIN {X 0,Y 587.363,Z 115.316,A -85,B 0,C 180,E1 -1628.255,E2 -1628.255} C_VEL
LIN {X 0,Y 587.346,Z 115.322,A -85,B 0,C 180,E1 -1631.134,E2 -1631.134} C_VEL
LIN {X 0,Y 587.362,Z 115.318,A -85,B 0,C 180,E1 -1634.26,E2 -1634.26} C_VEL
LIN {X 0,Y 587.348,Z 115.318,A -85,B 0,C 180,E1 -1637.406,E2 -1637.406} C_VEL
LIN {X 0,Y 587.309,Z 115.324,A -85,B 0,C 180,E1 -1638.308,E2 -1638.308} C_VEL
LIN {X 0,Y 586.666,Z 115.408,A -85,B 0,C 180,E1 -1638.88,E2 -1638.88} C_VEL
LIN {X 0,Y 583.841,Z 115.759,A -85,B 0,C 180,E1 -1639.809,E2 -1639.809} C_VEL
LIN {X 0,Y 581.429,Z 116.064,A -85,B 0,C 180,E1 -1640.556,E2 -1640.556} C_VEL
LIN {X 0,Y 580.376,Z 116.188,A -85,B 0,C 180,E1 -1641.132,E2 -1641.132} C_VEL
LIN {X 0,Y 580.281,Z 116.198,A -85,B 0,C 180,E1 -1641.328,E2 -1641.328} C_VEL
LIN {X 0,Y 580.276,Z 116.199,A -85,B 0,C 180,E1 -1643.558,E2 -1643.558} C_VEL
LIN {X 0,Y 580.291,Z 116.198,A -85,B 0,C 180,E1 -1645.849,E2 -1645.849} C_VEL
LIN {X 0,Y 580.301,Z 116.202,A -85,B 0,C 180,E1 -1648.185,E2 -1648.185} C_VEL
LIN {X 0,Y 580.29,Z 116.202,A -85,B 0,C 180,E1 -1650.696,E2 -1650.696} C_VEL
LIN {X 0,Y 580.302,Z 116.196,A -85,B 0,C 180,E1 -1653.317,E2 -1653.317} C_VEL
LIN {X 0,Y 580.34,Z 116.38,A -85,B 0,C 180,E1 -1655.488,E2 -1655.488} C_VEL
LIN {X 0,Y 580.324,Z 128.807,A -85,B 0,C 180,E1 -1657.87,E2 -1657.87} C_VEL
LIN {X 0,Y 580.262,Z 136.834,A -85,B 0,C 180,E1 -1659.393,E2 -1659.393} C_VEL
LIN {X 0,Y 580.928,Z 142.335,A -85,B 0,C 180,E1 -1659.489,E2 -1659.489} C_VEL
LIN {X 0,Y 580.787,Z 243.547,A -85,B 0,C 180,E1 -1660.764,E2 -1660.764} C_VEL
LIN {X 0,Y 580.688,Z 257.411,A -85,B 0,C 180,E1 -1661.096,E2 -1661.096} C_VEL
LIN {X 0,Y 580.631,Z 269.376,A -85,B 0,C 180,E1 -1661.52,E2 -1661.52} C_VEL
LIN {X 0,Y 580.528,Z 281.406,A -85,B 0,C 180,E1 -1662.096,E2 -1662.096} C_VEL
LIN {X 0,Y 580.46,Z 292.932,A -85,B 0,C 180,E1 -1662.808,E2 -1662.808} C_VEL
LIN {X 0,Y 580.376,Z 303.786,A -85,B 0,C 180,E1 -1663.649,E2 -1663.649} C_VEL
LIN {X 0,Y 580.269,Z 313.011,A -85,B 0,C 180,E1 -1664.537,E2 -1664.537} C_VEL
LIN {X 0,Y 580.193,Z 322.106,A -85,B 0,C 180,E1 -1665.617,E2 -1665.617} C_VEL
LIN {X 0,Y 580.156,Z 328.914,A -85,B 0,C 180,E1 -1666.622,E2 -1666.622} C_VEL
LIN {X 0,Y 580.123,Z 334.502,A -85,B 0,C 180,E1 -1667.646,E2 -1667.646} C_VEL
LIN {X 0,Y 580.048,Z 339.031,A -85,B 0,C 180,E1 -1668.695,E2 -1668.695} C_VEL
LIN {X 0,Y 580.062,Z 343.257,A -85,B 0,C 180,E1 -1670.048,E2 -1670.048} C_VEL
LIN {X 0,Y 580.014,Z 345.171,A -85,B 0,C 180,E1 -1670.944,E2 -1670.944} C_VEL
LIN {X 0,Y 580.018,Z 346.517,A -85,B 0,C 180,E1 -1671.961,E2 -1671.961} C_VEL
LIN {X 0,Y 580.03,Z 346.994,A -85,B 0,C 180,E1 -1673.101,E2 -1673.101} C_VEL
LIN {X 0,Y 580.042,Z 346.18,A -85,B 0,C 180,E1 -1674.438,E2 -1674.438} C_VEL
LIN {X 0,Y 580.049,Z 344.537,A -85,B 0,C 180,E1 -1675.477,E2 -1675.477} C_VEL
LIN {X 0,Y 580.071,Z 341.346,A -85,B 0,C 180,E1 -1676.719,E2 -1676.719} C_VEL
LIN {X 0,Y 580.093,Z 336.55,A -85,B 0,C 180,E1 -1678.002,E2 -1678.002} C_VEL
LIN {X 0,Y 580.127,Z 331.66,A -85,B 0,C 180,E1 -1678.994,E2 -1678.994} C_VEL
LIN {X 0,Y 580.159,Z 325.346,A -85,B 0,C 180,E1 -1680.02,E2 -1680.02} C_VEL
LIN {X 0,Y 580.235,Z 317.74,A -85,B 0,C 180,E1 -1681.021,E2 -1681.021} C_VEL
LIN {X 0,Y 580.307,Z 308.509,A -85,B 0,C 180,E1 -1682.009,E2 -1682.009} C_VEL
LIN {X 0,Y 580.398,Z 298.214,A -85,B 0,C 180,E1 -1682.897,E2 -1682.897} C_VEL
LIN {X 0,Y 580.494,Z 286.404,A -85,B 0,C 180,E1 -1683.706,E2 -1683.706} C_VEL
LIN {X 0,Y 580.591,Z 274.188,A -85,B 0,C 180,E1 -1684.358,E2 -1684.358} C_VEL
LIN {X 0,Y 580.677,Z 262.128,A -85,B 0,C 180,E1 -1684.842,E2 -1684.842} C_VEL
LIN {X 0,Y 580.761,Z 249.248,A -85,B 0,C 180,E1 -1685.209,E2 -1685.209} C_VEL
LIN {X 0,Y 580.839,Z 236.189,A -85,B 0,C 180,E1 -1685.436,E2 -1685.436} C_VEL
LIN {X 0,Y 580.875,Z 140.469,A -85,B 0,C 180,E1 -1686.625,E2 -1686.625} C_VEL
LIN {X 0,Y 580.295,Z 136.822,A -85,B 0,C 180,E1 -1686.699,E2 -1686.699} C_VEL
LIN {X 0,Y 580.353,Z 120.491,A -85,B 0,C 180,E1 -1689.81,E2 -1689.81} C_VEL
LIN {X 0,Y 580.326,Z 116.195,A -85,B 0,C 180,E1 -1690.667,E2 -1690.667} C_VEL
LIN {X 0,Y 580.268,Z 116.208,A -85,B 0,C 180,E1 -1693.825,E2 -1693.825} C_VEL
LIN {X 0,Y 580.324,Z 116.198,A -85,B 0,C 180,E1 -1695.983,E2 -1695.983} C_VEL
LIN {X 0,Y 580.306,Z 116.194,A -85,B 0,C 180,E1 -1698.827,E2 -1698.827} C_VEL
LIN {X 0,Y 580.327,Z 116.2,A -85,B 0,C 180,E1 -1701.644,E2 -1701.644} C_VEL
LIN {X 0,Y 580.32,Z 116.192,A -85,B 0,C 180,E1 -1704.44,E2 -1704.44} C_VEL
LIN {X 0,Y 580.339,Z 116.197,A -85,B 0,C 180,E1 -1707.224,E2 -1707.224} C_VEL
LIN {X 0,Y 580.353,Z 116.189,A -85,B 0,C 180,E1 -1710,E2 -1710} C_VEL
LIN {X 0,Y 580.328,Z 116.194,A -85,B 0,C 180,E1 -1712.777,E2 -1712.777} C_VEL
LIN {X 0,Y 580.333,Z 116.195,A -85,B 0,C 180,E1 -1715.56,E2 -1715.56} C_VEL
LIN {X 0,Y 580.309,Z 116.194,A -85,B 0,C 180,E1 -1718.356,E2 -1718.356} C_VEL
LIN {X 0,Y 580.301,Z 116.203,A -85,B 0,C 180,E1 -1721.191,E2 -1721.191} C_VEL
LIN {X 0,Y 580.325,Z 116.191,A -85,B 0,C 180,E1 -1724.017,E2 -1724.017} C_VEL
LIN {X 0,Y 580.313,Z 116.203,A -85,B 0,C 180,E1 -1726.914,E2 -1726.914} C_VEL
LIN {X 0,Y 580.286,Z 116.196,A -85,B 0,C 180,E1 -1729.823,E2 -1729.823} C_VEL
LIN {X 0,Y 580.269,Z 116.199,A -85,B 0,C 180,E1 -1732.053,E2 -1732.053} C_VEL
LIN {X 0,Y 580.305,Z 116.198,A -85,B 0,C 180,E1 -1735.08,E2 -1735.08} C_VEL
LIN {X 0,Y 580.298,Z 116.198,A -85,B 0,C 180,E1 -1738.185,E2 -1738.185} C_VEL
LIN {X 0,Y 580.28,Z 116.205,A -85,B 0,C 180,E1 -1740.694,E2 -1740.694} C_VEL
LIN {X 0,Y 580.283,Z 116.197,A -85,B 0,C 180,E1 -1743.313,E2 -1743.313} C_VEL
LIN {X 0,Y 580.244,Z 116.202,A -85,B 0,C 180,E1 -1745.756,E2 -1745.756} C_VEL
LIN {X 0,Y 580.286,Z 116.202,A -85,B 0,C 180,E1 -1748.146,E2 -1748.146} C_VEL
LIN {X 0,Y 580.297,Z 116.197,A -85,B 0,C 180,E1 -1750.843,E2 -1750.843} C_VEL
LIN {X 0,Y 580.278,Z 116.199,A -85,B 0,C 180,E1 -1753.658,E2 -1753.658} C_VEL
LIN {X 0,Y 580.275,Z 116.201,A -85,B 0,C 180,E1 -1756.609,E2 -1756.609} C_VEL
LIN {X 0,Y 580.298,Z 116.195,A -85,B 0,C 180,E1 -1759.157,E2 -1759.157} C_VEL
LIN {X 0,Y 580.289,Z 116.204,A -85,B 0,C 180,E1 -1761.927,E2 -1761.927} C_VEL
LIN {X 0,Y 580.277,Z 116.2,A -85,B 0,C 180,E1 -1764.455,E2 -1764.455} C_VEL
LIN {X 0,Y 580.289,Z 116.196,A -85,B 0,C 180,E1 -1766.975,E2 -1766.975} C_VEL
LIN {X 0,Y 580.304,Z 116.197,A -85,B 0,C 180,E1 -1769.426,E2 -1769.426} C_VEL
LIN {X 0,Y 580.295,Z 116.2,A -85,B 0,C 180,E1 -1772.141,E2 -1772.141} C_VEL
LIN {X 0,Y 580.32,Z 116.195,A -85,B 0,C 180,E1 -1775.27,E2 -1775.27} C_VEL
LIN {X 0,Y 580.273,Z 116.203,A -85,B 0,C 180,E1 -1777.948,E2 -1777.948} C_VEL
LIN {X 0,Y 580.317,Z 116.194,A -85,B 0,C 180,E1 -1780.914,E2 -1780.914} C_VEL
LIN {X 0,Y 580.277,Z 116.202,A -85,B 0,C 180,E1 -1783.826,E2 -1783.826} C_VEL
LIN {X 0,Y 580.323,Z 116.194,A -85,B 0,C 180,E1 -1785.983,E2 -1785.983} C_VEL
LIN {X 0,Y 580.303,Z 116.196,A -85,B 0,C 180,E1 -1788.827,E2 -1788.827} C_VEL
LIN {X 0,Y 580.333,Z 116.195,A -85,B 0,C 180,E1 -1791.644,E2 -1791.644} C_VEL
LIN {X 0,Y 580.326,Z 116.192,A -85,B 0,C 180,E1 -1794.44,E2 -1794.44} C_VEL
LIN {X 0,Y 580.345,Z 116.19,A -85,B 0,C 180,E1 -1797.918,E2 -1797.918} C_VEL
LIN {X 0,Y 580.357,Z 116.191,A -85,B 0,C 180,E1 -1800.694,E2 -1800.694} C_VEL
LIN {X 0,Y 580.284,Z 116.2,A -85,B 0,C 180,E1 -1803.472,E2 -1803.472} C_VEL
LIN {X 0,Y 580.33,Z 116.193,A -85,B 0,C 180,E1 -1805.56,E2 -1805.56} C_VEL
LIN {X 0,Y 580.326,Z 116.194,A -85,B 0,C 180,E1 -1808.356,E2 -1808.356} C_VEL
LIN {X 0,Y 580.299,Z 116.199,A -85,B 0,C 180,E1 -1811.191,E2 -1811.191} C_VEL
LIN {X 0,Y 580.324,Z 116.192,A -85,B 0,C 180,E1 -1814.017,E2 -1814.017} C_VEL
LIN {X 0,Y 580.311,Z 116.199,A -85,B 0,C 180,E1 -1816.914,E2 -1816.914} C_VEL
LIN {X 0,Y 580.304,Z 116.195,A -85,B 0,C 180,E1 -1819.823,E2 -1819.823} C_VEL
LIN {X 0,Y 580.294,Z 116.201,A -85,B 0,C 180,E1 -1822.803,E2 -1822.803} C_VEL
LIN {X 0,Y 580.306,Z 116.196,A -85,B 0,C 180,E1 -1825.08,E2 -1825.08} C_VEL
LIN {X 0,Y 580.299,Z 116.201,A -85,B 0,C 180,E1 -1828.186,E2 -1828.186} C_VEL
LIN {X 0,Y 580.287,Z 116.201,A -85,B 0,C 180,E1 -1830.695,E2 -1830.695} C_VEL
LIN {X 0,Y 580.304,Z 116.194,A -85,B 0,C 180,E1 -1833.317,E2 -1833.317} C_VEL
LIN {X 0,Y 580.245,Z 116.205,A -85,B 0,C 180,E1 -1835.757,E2 -1835.757} C_VEL
LIN {X 0,Y 580.291,Z 116.206,A -85,B 0,C 180,E1 -1838.146,E2 -1838.146} C_VEL
LIN {X 0,Y 580.301,Z 116.195,A -85,B 0,C 180,E1 -1840.844,E2 -1840.844} C_VEL
LIN {X 0,Y 580.28,Z 116.201,A -85,B 0,C 180,E1 -1843.658,E2 -1843.658} C_VEL
LIN {X 0,Y 580.278,Z 116.198,A -85,B 0,C 180,E1 -1846.61,E2 -1846.61} C_VEL
LIN {X 0,Y 580.301,Z 116.195,A -85,B 0,C 180,E1 -1849.157,E2 -1849.157} C_VEL
LIN {X 0,Y 580.293,Z 116.204,A -85,B 0,C 180,E1 -1851.927,E2 -1851.927} C_VEL
LIN {X 0,Y 580.252,Z 116.202,A -85,B 0,C 180,E1 -1854.453,E2 -1854.453} C_VEL
LIN {X 0,Y 580.292,Z 116.196,A -85,B 0,C 180,E1 -1856.975,E2 -1856.975} C_VEL
LIN {X 0,Y 580.297,Z 116.202,A -85,B 0,C 180,E1 -1859.425,E2 -1859.425} C_VEL
LIN {X 0,Y 580.3,Z 116.197,A -85,B 0,C 180,E1 -1862.141,E2 -1862.141} C_VEL
LIN {X 0,Y 580.324,Z 116.201,A -85,B 0,C 180,E1 -1865.27,E2 -1865.27} C_VEL
LIN {X 0,Y 580.351,Z 116.301,A -85,B 0,C 180,E1 -1865.924,E2 -1865.924} C_VEL
LIN {X 0,Y 580.983,Z 120.176,A -85,B 0,C 180,E1 -1866.472,E2 -1866.472} C_VEL
LIN {X 0,Y 580.833,Z 139.707,A -85,B 0,C 180,E1 -1869.087,E2 -1869.087} C_VEL
LIN {X 0,Y 580.719,Z 160.322,A -85,B 0,C 180,E1 -1871.842,E2 -1871.842} C_VEL
LIN {X 0,Y 580.484,Z 182.158,A -85,B 0,C 180,E1 -1874.732,E2 -1874.732} C_VEL
LIN {X 0,Y 580.401,Z 194.355,A -85,B 0,C 180,E1 -1876.331,E2 -1876.331} C_VEL
LIN {X 0,Y 580.963,Z 200.513,A -85,B 0,C 180,E1 -1876.423,E2 -1876.423} C_VEL
LIN {X 0,Y 580.809,Z 302.949,A -85,B 0,C 180,E1 -1877.708,E2 -1877.708} C_VEL
LIN {X 0,Y 580.727,Z 316.22,A -85,B 0,C 180,E1 -1878.017,E2 -1878.017} C_VEL
LIN {X 0,Y 580.653,Z 328.376,A -85,B 0,C 180,E1 -1878.436,E2 -1878.436} C_VEL
LIN {X 0,Y 580.579,Z 340.628,A -85,B 0,C 180,E1 -1879.009,E2 -1879.009} C_VEL
LIN {X 0,Y 580.441,Z 352.201,A -85,B 0,C 180,E1 -1879.712,E2 -1879.712} C_VEL
LIN {X 0,Y 580.345,Z 362.601,A -85,B 0,C 180,E1 -1880.503,E2 -1880.503} C_VEL
LIN {X 0,Y 580.271,Z 371.113,A -85,B 0,C 180,E1 -1881.292,E2 -1881.292} C_VEL
LIN {X 0,Y 580.222,Z 378.961,A -85,B 0,C 180,E1 -1882.168,E2 -1882.168} C_VEL
LIN {X 0,Y 580.154,Z 386.651,A -85,B 0,C 180,E1 -1883.222,E2 -1883.222} C_VEL
LIN {X 0,Y 580.139,Z 393.68,A -85,B 0,C 180,E1 -1884.438,E2 -1884.438} C_VEL
LIN {X 0,Y 580.108,Z 398.372,A -85,B 0,C 180,E1 -1885.483,E2 -1885.483} C_VEL
LIN {X 0,Y 580.123,Z 401.957,A -85,B 0,C 180,E1 -1886.527,E2 -1886.527} C_VEL
LIN {X 0,Y 580.043,Z 403.808,A -85,B 0,C 180,E1 -1887.222,E2 -1887.222} C_VEL
LIN {X 0,Y 580.04,Z 405.198,A -85,B 0,C 180,E1 -1887.917,E2 -1887.917} C_VEL
LIN {X 0,Y 580.04,Z 406.785,A -85,B 0,C 180,E1 -1889.306,E2 -1889.306} C_VEL
LIN {X 0,Y 580.037,Z 407,A -85,B 0,C 180,E1 -1890,E2 -1890} C_VEL
LIN {X 0,Y 580.047,Z 406.186,A -85,B 0,C 180,E1 -1891.389,E2 -1891.389} C_VEL
LIN {X 0,Y 580.04,Z 405.2,A -85,B 0,C 180,E1 -1892.083,E2 -1892.083} C_VEL
LIN {X 0,Y 580.043,Z 403.81,A -85,B 0,C 180,E1 -1892.778,E2 -1892.778} C_VEL
LIN {X 0,Y 580.11,Z 400.896,A -85,B 0,C 180,E1 -1893.821,E2 -1893.821} C_VEL
LIN {X 0,Y 580.053,Z 396.949,A -85,B 0,C 180,E1 -1894.865,E2 -1894.865} C_VEL
LIN {X 0,Y 580.139,Z 390.877,A -85,B 0,C 180,E1 -1896.085,E2 -1896.085} C_VEL
LIN {X 0,Y 580.184,Z 384.238,A -85,B 0,C 180,E1 -1897.132,E2 -1897.132} C_VEL
LIN {X 0,Y 580.25,Z 375.991,A -85,B 0,C 180,E1 -1898.182,E2 -1898.182} C_VEL
LIN {X 0,Y 580.308,Z 367.539,A -85,B 0,C 180,E1 -1899.058,E2 -1899.058} C_VEL
LIN {X 0,Y 580.422,Z 357.099,A -85,B 0,C 180,E1 -1899.936,E2 -1899.936} C_VEL
LIN {X 0,Y 580.506,Z 346.756,A -85,B 0,C 180,E1 -1900.639,E2 -1900.639} C_VEL
LIN {X 0,Y 580.596,Z 335.248,A -85,B 0,C 180,E1 -1901.264,E2 -1901.264} C_VEL
LIN {X 0,Y 580.682,Z 322.475,A -85,B 0,C 180,E1 -1901.785,E2 -1901.785} C_VEL
LIN {X 0,Y 580.777,Z 309.438,A -85,B 0,C 180,E1 -1902.159,E2 -1902.159} C_VEL
LIN {X 0,Y 580.839,Z 297.092,A -85,B 0,C 180,E1 -1902.38,E2 -1902.38} C_VEL
LIN {X 0,Y 580.802,Z 197.166,A -85,B 0,C 180,E1 -1903.623,E2 -1903.623} C_VEL
LIN {X 0,Y 580.407,Z 194.27,A -85,B 0,C 180,E1 -1903.68,E2 -1903.68} C_VEL
LIN {X 0,Y 580.602,Z 171.24,A -85,B 0,C 180,E1 -1906.707,E2 -1906.707} C_VEL
LIN {X 0,Y 580.73,Z 152.006,A -85,B 0,C 180,E1 -1909.272,E2 -1909.272} C_VEL
LIN {X 0,Y 580.877,Z 132.636,A -85,B 0,C 180,E1 -1911.841,E2 -1911.841} C_VEL
LIN {X 0,Y 580.954,Z 119.956,A -85,B 0,C 180,E1 -1913.529,E2 -1913.529} C_VEL
LIN {X 0,Y 580.318,Z 116.202,A -85,B 0,C 180,E1 -1914.078,E2 -1914.078} C_VEL
LIN {X 0,Y 580.279,Z 116.206,A -85,B 0,C 180,E1 -1916.623,E2 -1916.623} C_VEL
LIN {X 0,Y 580.303,Z 116.195,A -85,B 0,C 180,E1 -1919.309,E2 -1919.309} C_VEL
LIN {X 0,Y 580.301,Z 116.202,A -85,B 0,C 180,E1 -1922.2,E2 -1922.2} C_VEL
LIN {X 0,Y 580.29,Z 116.2,A -85,B 0,C 180,E1 -1924.696,E2 -1924.696} C_VEL
LIN {X 0,Y 580.3,Z 116.195,A -85,B 0,C 180,E1 -1927.268,E2 -1927.268} C_VEL
LIN {X 0,Y 580.298,Z 116.204,A -85,B 0,C 180,E1 -1930.271,E2 -1930.271} C_VEL
LIN {X 0,Y 580.278,Z 116.2,A -85,B 0,C 180,E1 -1932.706,E2 -1932.706} C_VEL
LIN {X 0,Y 580.27,Z 116.202,A -85,B 0,C 180,E1 -1935.609,E2 -1935.609} C_VEL
LIN {X 0,Y 580.314,Z 116.199,A -85,B 0,C 180,E1 -1938.234,E2 -1938.234} C_VEL
LIN {X 0,Y 580.289,Z 116.196,A -85,B 0,C 180,E1 -1940.966,E2 -1940.966} C_VEL
LIN {X 0,Y 580.267,Z 116.204,A -85,B 0,C 180,E1 -1943.596,E2 -1943.596} C_VEL
LIN {X 0,Y 580.315,Z 116.197,A -85,B 0,C 180,E1 -1946.145,E2 -1946.145} C_VEL
LIN {X 0,Y 580.281,Z 116.197,A -85,B 0,C 180,E1 -1948.615,E2 -1948.615} C_VEL
LIN {X 0,Y 580.291,Z 116.196,A -85,B 0,C 180,E1 -1951.024,E2 -1951.024} C_VEL
LIN {X 0,Y 580.291,Z 116.205,A -85,B 0,C 180,E1 -1953.665,E2 -1953.665} C_VEL
LIN {X 0,Y 580.296,Z 116.204,A -85,B 0,C 180,E1 -1955.683,E2 -1955.683} C_VEL
LIN {X 0,Y 580.284,Z 116.197,A -85,B 0,C 180,E1 -1958.694,E2 -1958.694} C_VEL
LIN {X 0,Y 580.318,Z 116.194,A -85,B 0,C 180,E1 -1960.914,E2 -1960.914} C_VEL
LIN {X 0,Y 580.277,Z 116.201,A -85,B 0,C 180,E1 -1963.825,E2 -1963.825} C_VEL
LIN {X 0,Y 580.323,Z 116.193,A -85,B 0,C 180,E1 -1965.983,E2 -1965.983} C_VEL
LIN {X 0,Y 580.303,Z 116.197,A -85,B 0,C 180,E1 -1968.827,E2 -1968.827} C_VEL
LIN {X 0,Y 580.332,Z 116.194,A -85,B 0,C 180,E1 -1971.644,E2 -1971.644} C_VEL
LIN {X 0,Y 580.327,Z 116.192,A -85,B 0,C 180,E1 -1974.44,E2 -1974.44} C_VEL
LIN {X 0,Y 580.345,Z 116.19,A -85,B 0,C 180,E1 -1977.918,E2 -1977.918} C_VEL
LIN {X 0,Y 580.357,Z 116.192,A -85,B 0,C 180,E1 -1980.694,E2 -1980.694} C_VEL
LIN {X 0,Y 580.283,Z 116.2,A -85,B 0,C 180,E1 -1983.472,E2 -1983.472} C_VEL
LIN {X 0,Y 580.329,Z 116.192,A -85,B 0,C 180,E1 -1985.56,E2 -1985.56} C_VEL
LIN {X 0,Y 580.326,Z 116.194,A -85,B 0,C 180,E1 -1988.356,E2 -1988.356} C_VEL
LIN {X 0,Y 580.297,Z 116.199,A -85,B 0,C 180,E1 -1991.191,E2 -1991.191} C_VEL
LIN {X 0,Y 580.323,Z 116.193,A -85,B 0,C 180,E1 -1994.017,E2 -1994.017} C_VEL
LIN {X 0,Y 580.31,Z 116.2,A -85,B 0,C 180,E1 -1996.914,E2 -1996.914} C_VEL
LIN {X 0,Y 580.303,Z 116.195,A -85,B 0,C 180,E1 -1999.822,E2 -1999.822} C_VEL
LIN {X 0,Y 580.281,Z 116.198,A -85,B 0,C 180,E1 -2001.328,E2 -2001.328} C_VEL
LIN {X 0,Y 579.585,Z 116.286,A -85,B 0,C 180,E1 -2001.907,E2 -2001.907} C_VEL
LIN {X 0,Y 576.708,Z 116.648,A -85,B 0,C 180,E1 -2002.847,E2 -2002.847} C_VEL
LIN {X 0,Y 574.313,Z 116.944,A -85,B 0,C 180,E1 -2003.603,E2 -2003.603} C_VEL
LIN {X 0,Y 573.314,Z 117.071,A -85,B 0,C 180,E1 -2004.187,E2 -2004.187} C_VEL
LIN {X 0,Y 573.247,Z 117.079,A -85,B 0,C 180,E1 -2004.384,E2 -2004.384} C_VEL
LIN {X 0,Y 573.249,Z 117.076,A -85,B 0,C 180,E1 -2006.976,E2 -2006.976} C_VEL
LIN {X 0,Y 573.245,Z 117.074,A -85,B 0,C 180,E1 -2009.488,E2 -2009.488} C_VEL
LIN {X 0,Y 573.255,Z 117.082,A -85,B 0,C 180,E1 -2012.229,E2 -2012.229} C_VEL
LIN {X 0,Y 573.272,Z 117.076,A -85,B 0,C 180,E1 -2014.777,E2 -2014.777} C_VEL
LIN {X 0,Y 573.298,Z 117.232,A -85,B 0,C 180,E1 -2015.45,E2 -2015.45} C_VEL
LIN {X 0,Y 573.296,Z 127.662,A -85,B 0,C 180,E1 -2017.458,E2 -2017.458} C_VEL
LIN {X 0,Y 573.22,Z 136.883,A -85,B 0,C 180,E1 -2019.231,E2 -2019.231} C_VEL
LIN {X 0,Y 574.025,Z 143.244,A -85,B 0,C 180,E1 -2019.335,E2 -2019.335} C_VEL
LIN {X 0,Y 573.876,Z 242.785,A -85,B 0,C 180,E1 -2020.599,E2 -2020.599} C_VEL
LIN {X 0,Y 573.758,Z 256.193,A -85,B 0,C 180,E1 -2020.914,E2 -2020.914} C_VEL
LIN {X 0,Y 573.676,Z 268.965,A -85,B 0,C 180,E1 -2021.362,E2 -2021.362} C_VEL
LIN {X 0,Y 573.562,Z 280.636,A -85,B 0,C 180,E1 -2021.918,E2 -2021.918} C_VEL
LIN {X 0,Y 573.458,Z 292.705,A -85,B 0,C 180,E1 -2022.666,E2 -2022.666} C_VEL
LIN {X 0,Y 573.334,Z 303.582,A -85,B 0,C 180,E1 -2023.514,E2 -2023.514} C_VEL
LIN {X 0,Y 573.224,Z 313.654,A -85,B 0,C 180,E1 -2024.502,E2 -2024.502} C_VEL
LIN {X 0,Y 573.114,Z 321.872,A -85,B 0,C 180,E1 -2025.494,E2 -2025.494} C_VEL
LIN {X 0,Y 573.065,Z 329.393,A -85,B 0,C 180,E1 -2026.625,E2 -2026.625} C_VEL
LIN {X 0,Y 573.044,Z 335.561,A -85,B 0,C 180,E1 -2027.81,E2 -2027.81} C_VEL
LIN {X 0,Y 572.983,Z 340.255,A -85,B 0,C 180,E1 -2028.989,E2 -2028.989} C_VEL
LIN {X 0,Y 572.935,Z 344.096,A -85,B 0,C 180,E1 -2030.367,E2 -2030.367} C_VEL
LIN {X 0,Y 572.927,Z 346.285,A -85,B 0,C 180,E1 -2031.728,E2 -2031.728} C_VEL
LIN {X 0,Y 572.951,Z 347,A -85,B 0,C 180,E1 -2033.055,E2 -2033.055} C_VEL
LIN {X 0,Y 572.923,Z 346.575,A -85,B 0,C 180,E1 -2034.058,E2 -2034.058} C_VEL
LIN {X 0,Y 572.961,Z 345.012,A -85,B 0,C 180,E1 -2035.268,E2 -2035.268} C_VEL
LIN {X 0,Y 572.987,Z 342.088,A -85,B 0,C 180,E1 -2036.518,E2 -2036.518} C_VEL
LIN {X 0,Y 572.994,Z 337.586,A -85,B 0,C 180,E1 -2037.813,E2 -2037.813} C_VEL
LIN {X 0,Y 573.054,Z 332.033,A -85,B 0,C 180,E1 -2038.997,E2 -2038.997} C_VEL
LIN {X 0,Y 573.106,Z 324.664,A -85,B 0,C 180,E1 -2040.204,E2 -2040.204} C_VEL
LIN {X 0,Y 573.162,Z 316.807,A -85,B 0,C 180,E1 -2041.231,E2 -2041.231} C_VEL
LIN {X 0,Y 573.275,Z 307.334,A -85,B 0,C 180,E1 -2042.235,E2 -2042.235} C_VEL
LIN {X 0,Y 573.39,Z 298.048,A -85,B 0,C 180,E1 -2043.031,E2 -2043.031} C_VEL
LIN {X 0,Y 573.486,Z 286.667,A -85,B 0,C 180,E1 -2043.821,E2 -2043.821} C_VEL
LIN {X 0,Y 573.633,Z 274.941,A -85,B 0,C 180,E1 -2044.462,E2 -2044.462} C_VEL
LIN {X 0,Y 573.721,Z 262.175,A -85,B 0,C 180,E1 -2044.985,E2 -2044.985} C_VEL
LIN {X 0,Y 573.86,Z 248.936,A -85,B 0,C 180,E1 -2045.366,E2 -2045.366} C_VEL
LIN {X 0,Y 573.924,Z 236.114,A -85,B 0,C 180,E1 -2045.589,E2 -2045.589} C_VEL
LIN {X 0,Y 573.925,Z 140.996,A -85,B 0,C 180,E1 -2046.786,E2 -2046.786} C_VEL
LIN {X 0,Y 573.237,Z 136.9,A -85,B 0,C 180,E1 -2046.855,E2 -2046.855} C_VEL
LIN {X 0,Y 573.338,Z 121.007,A -85,B 0,C 180,E1 -2049.927,E2 -2049.927} C_VEL
LIN {X 0,Y 573.282,Z 117.073,A -85,B 0,C 180,E1 -2050.727,E2 -2050.727} C_VEL
LIN {X 0,Y 573.242,Z 117.083,A -85,B 0,C 180,E1 -2053.622,E2 -2053.622} C_VEL
LIN {X 0,Y 573.272,Z 117.079,A -85,B 0,C 180,E1 -2055.807,E2 -2055.807} C_VEL
LIN {X 0,Y 573.264,Z 117.071,A -85,B 0,C 180,E1 -2058.745,E2 -2058.745} C_VEL
LIN {X 0,Y 573.282,Z 117.079,A -85,B 0,C 180,E1 -2061.541,E2 -2061.541} C_VEL
LIN {X 0,Y 573.29,Z 117.068,A -85,B 0,C 180,E1 -2064.372,E2 -2064.372} C_VEL
LIN {X 0,Y 573.316,Z 117.067,A -85,B 0,C 180,E1 -2067.892,E2 -2067.892} C_VEL
LIN {X 0,Y 573.322,Z 117.065,A -85,B 0,C 180,E1 -2070.702,E2 -2070.702} C_VEL
LIN {X 0,Y 573.297,Z 117.07,A -85,B 0,C 180,E1 -2072.811,E2 -2072.811} C_VEL
LIN {X 0,Y 573.299,Z 117.07,A -85,B 0,C 180,E1 -2075.628,E2 -2075.628} C_VEL
LIN {X 0,Y 573.254,Z 117.073,A -85,B 0,C 180,E1 -2078.46,E2 -2078.46} C_VEL
LIN {X 0,Y 573.273,Z 117.076,A -85,B 0,C 180,E1 -2081.312,E2 -2081.312} C_VEL
LIN {X 0,Y 573.282,Z 117.071,A -85,B 0,C 180,E1 -2084.424,E2 -2084.424} C_VEL
LIN {X 0,Y 573.258,Z 117.079,A -85,B 0,C 180,E1 -2087.112,E2 -2087.112} C_VEL
LIN {X 0,Y 573.241,Z 117.075,A -85,B 0,C 180,E1 -2090.077,E2 -2090.077} C_VEL
LIN {X 0,Y 573.234,Z 117.078,A -85,B 0,C 180,E1 -2092.338,E2 -2092.338} C_VEL
LIN {X 0,Y 573.248,Z 117.074,A -85,B 0,C 180,E1 -2095.41,E2 -2095.41} C_VEL
LIN {X 0,Y 573.251,Z 117.074,A -85,B 0,C 180,E1 -2098.029,E2 -2098.029} C_VEL
LIN {X 0,Y 573.226,Z 117.081,A -85,B 0,C 180,E1 -2100.882,E2 -2100.882} C_VEL
LIN {X 0,Y 573.24,Z 117.074,A -85,B 0,C 180,E1 -2103.521,E2 -2103.521} C_VEL
LIN {X 0,Y 573.213,Z 117.081,A -85,B 0,C 180,E1 -2106.051,E2 -2106.051} C_VEL
LIN {X 0,Y 573.241,Z 117.079,A -85,B 0,C 180,E1 -2108.701,E2 -2108.701} C_VEL
LIN {X 0,Y 573.242,Z 117.075,A -85,B 0,C 180,E1 -2111.594,E2 -2111.594} C_VEL
LIN {X 0,Y 573.234,Z 117.083,A -85,B 0,C 180,E1 -2114.333,E2 -2114.333} C_VEL
LIN {X 0,Y 573.238,Z 117.075,A -85,B 0,C 180,E1 -2117.358,E2 -2117.358} C_VEL
LIN {X 0,Y 573.246,Z 117.078,A -85,B 0,C 180,E1 -2120.393,E2 -2120.393} C_VEL
LIN {X 0,Y 573.251,Z 117.073,A -85,B 0,C 180,E1 -2123.078,E2 -2123.078} C_VEL
LIN {X 0,Y 573.265,Z 117.076,A -85,B 0,C 180,E1 -2125.671,E2 -2125.671} C_VEL
LIN {X 0,Y 573.242,Z 117.079,A -85,B 0,C 180,E1 -2128.185,E2 -2128.185} C_VEL
LIN {X 0,Y 573.266,Z 117.071,A -85,B 0,C 180,E1 -2130.634,E2 -2130.634} C_VEL
LIN {X 0,Y 573.235,Z 117.08,A -85,B 0,C 180,E1 -2133.507,E2 -2133.507} C_VEL
LIN {X 0,Y 573.226,Z 117.079,A -85,B 0,C 180,E1 -2136.134,E2 -2136.134} C_VEL
LIN {X 0,Y 573.249,Z 117.076,A -85,B 0,C 180,E1 -2139.174,E2 -2139.174} C_VEL
LIN {X 0,Y 573.227,Z 117.083,A -85,B 0,C 180,E1 -2141.412,E2 -2141.412} C_VEL
LIN {X 0,Y 573.249,Z 117.081,A -85,B 0,C 180,E1 -2143.622,E2 -2143.622} C_VEL
LIN {X 0,Y 573.271,Z 117.075,A -85,B 0,C 180,E1 -2145.807,E2 -2145.807} C_VEL
LIN {X 0,Y 573.261,Z 117.073,A -85,B 0,C 180,E1 -2148.745,E2 -2148.745} C_VEL
LIN {X 0,Y 573.289,Z 117.074,A -85,B 0,C 180,E1 -2151.541,E2 -2151.541} C_VEL
LIN {X 0,Y 573.295,Z 117.067,A -85,B 0,C 180,E1 -2154.372,E2 -2154.372} C_VEL
LIN {X 0,Y 573.315,Z 117.066,A -85,B 0,C 180,E1 -2157.893,E2 -2157.893} C_VEL
LIN {X 0,Y 573.328,Z 117.067,A -85,B 0,C 180,E1 -2160.703,E2 -2160.703} C_VEL
LIN {X 0,Y 573.302,Z 117.073,A -85,B 0,C 180,E1 -2162.811,E2 -2162.811} C_VEL
LIN {X 0,Y 573.297,Z 117.068,A -85,B 0,C 180,E1 -2165.628,E2 -2165.628} C_VEL
LIN {X 0,Y 573.282,Z 117.072,A -85,B 0,C 180,E1 -2168.46,E2 -2168.46} C_VEL
LIN {X 0,Y 573.271,Z 117.073,A -85,B 0,C 180,E1 -2171.312,E2 -2171.312} C_VEL
LIN {X 0,Y 573.28,Z 117.074,A -85,B 0,C 180,E1 -2174.425,E2 -2174.425} C_VEL
LIN {X 0,Y 573.257,Z 117.075,A -85,B 0,C 180,E1 -2177.112,E2 -2177.112} C_VEL
LIN {X 0,Y 573.252,Z 117.075,A -85,B 0,C 180,E1 -2180.077,E2 -2180.077} C_VEL
LIN {X 0,Y 573.234,Z 117.077,A -85,B 0,C 180,E1 -2183.1,E2 -2183.1} C_VEL
LIN {X 0,Y 573.254,Z 117.072,A -85,B 0,C 180,E1 -2185.41,E2 -2185.41} C_VEL
LIN {X 0,Y 573.251,Z 117.077,A -85,B 0,C 180,E1 -2188.029,E2 -2188.029} C_VEL
LIN {X 0,Y 573.232,Z 117.077,A -85,B 0,C 180,E1 -2190.883,E2 -2190.883} C_VEL
LIN {X 0,Y 573.262,Z 117.072,A -85,B 0,C 180,E1 -2193.524,E2 -2193.524} C_VEL
LIN {X 0,Y 573.214,Z 117.085,A -85,B 0,C 180,E1 -2196.052,E2 -2196.052} C_VEL
LIN {X 0,Y 573.25,Z 117.075,A -85,B 0,C 180,E1 -2198.701,E2 -2198.701} C_VEL
LIN {X 0,Y 573.254,Z 117.075,A -85,B 0,C 180,E1 -2201.596,E2 -2201.596} C_VEL
LIN {X 0,Y 573.236,Z 117.079,A -85,B 0,C 180,E1 -2204.334,E2 -2204.334} C_VEL
LIN {X 0,Y 573.241,Z 117.076,A -85,B 0,C 180,E1 -2207.359,E2 -2207.359} C_VEL
LIN {X 0,Y 573.248,Z 117.075,A -85,B 0,C 180,E1 -2210.393,E2 -2210.393} C_VEL
LIN {X 0,Y 573.254,Z 117.073,A -85,B 0,C 180,E1 -2213.078,E2 -2213.078} C_VEL
LIN {X 0,Y 573.268,Z 117.08,A -85,B 0,C 180,E1 -2215.672,E2 -2215.672} C_VEL
LIN {X 0,Y 573.243,Z 117.076,A -85,B 0,C 180,E1 -2218.185,E2 -2218.185} C_VEL
LIN {X 0,Y 573.266,Z 117.072,A -85,B 0,C 180,E1 -2220.634,E2 -2220.634} C_VEL
LIN {X 0,Y 573.253,Z 117.076,A -85,B 0,C 180,E1 -2223.024,E2 -2223.024} C_VEL
LIN {X 0,Y 573.303,Z 117.193,A -85,B 0,C 180,E1 -2225.777,E2 -2225.777} C_VEL
LIN {X 0,Y 574.045,Z 122.072,A -85,B 0,C 180,E1 -2226.475,E2 -2226.475} C_VEL
LIN {X 0,Y 573.867,Z 140.935,A -85,B 0,C 180,E1 -2229.03,E2 -2229.03} C_VEL
LIN {X 0,Y 573.761,Z 161.65,A -85,B 0,C 180,E1 -2231.799,E2 -2231.799} C_VEL
LIN {X 0,Y 573.473,Z 183.522,A -85,B 0,C 180,E1 -2234.723,E2 -2234.723} C_VEL
LIN {X 0,Y 573.41,Z 194.355,A -85,B 0,C 180,E1 -2236.161,E2 -2236.161} C_VEL
LIN {X 0,Y 574.057,Z 200.513,A -85,B 0,C 180,E1 -2236.256,E2 -2236.256} C_VEL
LIN {X 0,Y 573.886,Z 302.949,A -85,B 0,C 180,E1 -2237.558,E2 -2237.558} C_VEL
LIN {X 0,Y 573.778,Z 316.22,A -85,B 0,C 180,E1 -2237.869,E2 -2237.869} C_VEL
LIN {X 0,Y 573.689,Z 329.497,A -85,B 0,C 180,E1 -2238.339,E2 -2238.339} C_VEL
LIN {X 0,Y 573.586,Z 340.67,A -85,B 0,C 180,E1 -2238.876,E2 -2238.876} C_VEL
LIN {X 0,Y 573.428,Z 352.199,A -85,B 0,C 180,E1 -2239.585,E2 -2239.585} C_VEL
LIN {X 0,Y 573.333,Z 362.603,A -85,B 0,C 180,E1 -2240.386,E2 -2240.386} C_VEL
LIN {X 0,Y 573.241,Z 371.113,A -85,B 0,C 180,E1 -2241.185,E2 -2241.185} C_VEL
LIN {X 0,Y 573.161,Z 378.961,A -85,B 0,C 180,E1 -2242.071,E2 -2242.071} C_VEL
LIN {X 0,Y 573.073,Z 386.955,A -85,B 0,C 180,E1 -2243.185,E2 -2243.185} C_VEL
LIN {X 0,Y 573.07,Z 393.68,A -85,B 0,C 180,E1 -2244.37,E2 -2244.37} C_VEL
LIN {X 0,Y 573.028,Z 398.372,A -85,B 0,C 180,E1 -2245.428,E2 -2245.428} C_VEL
LIN {X 0,Y 573.022,Z 401.958,A -85,B 0,C 180,E1 -2246.484,E2 -2246.484} C_VEL
LIN {X 0,Y 572.959,Z 403.808,A -85,B 0,C 180,E1 -2247.188,E2 -2247.188} C_VEL
LIN {X 0,Y 572.946,Z 406.185,A -85,B 0,C 180,E1 -2248.594,E2 -2248.594} C_VEL
LIN {X 0,Y 572.938,Z 407,A -85,B 0,C 180,E1 -2250,E2 -2250} C_VEL
LIN {X 0,Y 572.946,Z 406.186,A -85,B 0,C 180,E1 -2251.406,E2 -2251.406} C_VEL
LIN {X 0,Y 572.94,Z 405.199,A -85,B 0,C 180,E1 -2252.109,E2 -2252.109} C_VEL
LIN {X 0,Y 572.959,Z 403.81,A -85,B 0,C 180,E1 -2252.812,E2 -2252.812} C_VEL
LIN {X 0,Y 573.015,Z 400.896,A -85,B 0,C 180,E1 -2253.868,E2 -2253.868} C_VEL
LIN {X 0,Y 572.963,Z 396.949,A -85,B 0,C 180,E1 -2254.926,E2 -2254.926} C_VEL
LIN {X 0,Y 573.065,Z 390.877,A -85,B 0,C 180,E1 -2256.16,E2 -2256.16} C_VEL
LIN {X 0,Y 573.119,Z 384.237,A -85,B 0,C 180,E1 -2257.221,E2 -2257.221} C_VEL
LIN {X 0,Y 573.201,Z 375.992,A -85,B 0,C 180,E1 -2258.283,E2 -2258.283} C_VEL
LIN {X 0,Y 573.287,Z 367.54,A -85,B 0,C 180,E1 -2259.17,E2 -2259.17} C_VEL
LIN {X 0,Y 573.427,Z 357.097,A -85,B 0,C 180,E1 -2260.058,E2 -2260.058} C_VEL
LIN {X 0,Y 573.543,Z 345.433,A -85,B 0,C 180,E1 -2260.853,E2 -2260.853} C_VEL
LIN {X 0,Y 573.651,Z 334.31,A -85,B 0,C 180,E1 -2261.446,E2 -2261.446} C_VEL
LIN {X 0,Y 573.745,Z 321.172,A -85,B 0,C 180,E1 -2261.974,E2 -2261.974} C_VEL
LIN {X 0,Y 573.874,Z 308.522,A -85,B 0,C 180,E1 -2262.33,E2 -2262.33} C_VEL
LIN {X 0,Y 573.94,Z 295.318,A -85,B 0,C 180,E1 -2262.553,E2 -2262.553} C_VEL
LIN {X 0,Y 573.915,Z 197.959,A -85,B 0,C 180,E1 -2263.78,E2 -2263.78} C_VEL
LIN {X 0,Y 573.414,Z 194.27,A -85,B 0,C 180,E1 -2263.85,E2 -2263.85} C_VEL
LIN {X 0,Y 573.604,Z 172.627,A -85,B 0,C 180,E1 -2266.731,E2 -2266.731} C_VEL
LIN {X 0,Y 573.717,Z 156.043,A -85,B 0,C 180,E1 -2268.943,E2 -2268.943} C_VEL
LIN {X 0,Y 573.853,Z 139.549,A -85,B 0,C 180,E1 -2271.134,E2 -2271.134} C_VEL
LIN {X 0,Y 574.012,Z 121.748,A -85,B 0,C 180,E1 -2273.525,E2 -2273.525} C_VEL
LIN {X 0,Y 573.277,Z 117.08,A -85,B 0,C 180,E1 -2274.2,E2 -2274.2} C_VEL
LIN {X 0,Y 573.253,Z 117.077,A -85,B 0,C 180,E1 -2276.976,E2 -2276.976} C_VEL
LIN {X 0,Y 573.248,Z 117.075,A -85,B 0,C 180,E1 -2279.488,E2 -2279.488} C_VEL
LIN {X 0,Y 573.256,Z 117.078,A -85,B 0,C 180,E1 -2282.645,E2 -2282.645} C_VEL
LIN {X 0,Y 573.208,Z 117.079,A -85,B 0,C 180,E1 -2285.188,E2 -2285.188} C_VEL
LIN {X 0,Y 573.237,Z 117.079,A -85,B 0,C 180,E1 -2287.807,E2 -2287.807} C_VEL
LIN {X 0,Y 573.271,Z 117.075,A -85,B 0,C 180,E1 -2290.528,E2 -2290.528} C_VEL
LIN {X 0,Y 573.245,Z 117.078,A -85,B 0,C 180,E1 -2293.669,E2 -2293.669} C_VEL
LIN {X 0,Y 573.24,Z 117.077,A -85,B 0,C 180,E1 -2296.641,E2 -2296.641} C_VEL
LIN {X 0,Y 573.274,Z 117.073,A -85,B 0,C 180,E1 -2299.477,E2 -2299.477} C_VEL
LIN {X 0,Y 573.236,Z 117.08,A -85,B 0,C 180,E1 -2302.192,E2 -2302.192} C_VEL
LIN {X 0,Y 573.234,Z 117.076,A -85,B 0,C 180,E1 -2305.228,E2 -2305.228} C_VEL
LIN {X 0,Y 573.252,Z 117.082,A -85,B 0,C 180,E1 -2307.771,E2 -2307.771} C_VEL
